Yaskawa INFORM job: SKRZYNIA_5240_0_STOPNI_2OBR.JBI

/JOB
//NAME SKRZYNIA_5240_0_STOPNI_2OBR
///FOLDERNAME 02-SKRZYNIE_JOBS
//POS
///NPOS 621,621,0,54,0,0
///TOOL 0
///POSTYPE PULSE
///PULSE
C00000=1055,-24125,84372,288,19725,204
C00001=0,-15438,65714,0,-68532,0
C00002=4718,-16587,59952,3396,-65485,-935
C00003=32997,-21499,42555,27623,-61436,21376
C00004=31759,-20688,42932,26837,-60850,21559
C00005=28987,-21156,42712,24818,-60442,22222
C00006=33447,-21964,42352,27886,-61721,21330
C00007=37687,-23357,41794,30651,-63289,20620
C00008=38979,-19018,48057,32961,-64962,20678
C00009=37261,-18075,48526,31902,-64209,20901
C00010=35830,-17198,48994,31015,-63571,21092
C00011=34080,-17614,48768,29780,-63290,21485
C00012=37261,-18075,48526,31902,-64209,20901
C00013=47373,-21912,40596,41149,-66086,26950
C00014=0,-15438,65714,0,-68532,0
C00015=4718,-16587,59952,3396,-65485,-935
C00016=32997,-21499,42555,27623,-61436,21376
C00017=31759,-20688,42932,26837,-60850,21559
C00018=28987,-21156,42712,24818,-60442,22222
C00019=33447,-21964,42352,27886,-61721,21330
C00020=37687,-23357,41794,30651,-63289,20620
C00021=38979,-19018,48057,32961,-64962,20678
C00022=37261,-18075,48526,31902,-64209,20901
C00023=35830,-17198,48994,31015,-63571,21092
C00024=34080,-17614,48768,29780,-63290,21485
C00025=37261,-18075,48526,31902,-64209,20901
C00026=47373,-21912,40596,41149,-66086,26950
C00027=45033,-20851,41104,39798,-65001,27223
C00028=42790,-19693,41704,38494,-63946,27495
C00029=41070,-20182,41442,37324,-63566,27891
C00030=45033,-20851,41104,39798,-65001,27223
C00031=45033,-20851,41104,39798,-65001,27223
C00032=59624,-29540,14278,64846,-60867,16042
C00033=57357,-28542,14780,63940,-59509,16120
C00034=56188,-29140,14476,63237,-58995,16387
C00035=59588,-29370,14363,64862,-60819,16012
C00036=62924,-29779,15793,65870,-63073,16252
C00037=59724,-28781,16276,64511,-61238,16415
C00038=57764,-27936,16704,63709,-60078,16488
C00039=56408,-28589,16373,62897,-59486,16787
C00040=59724,-28781,16276,64511,-61238,16415
C00041=87562,-48087,-13810,78020,-75252,11220
C00042=10104,-46603,4759,11228,-37390,-5046
C00043=0,-52280,40443,0,6876,0
C00044=1529,-42140,58025,-5964,2417,3265
C00045=0,-38374,23626,-1605,-51738,268
C00046=45044,-23015,37260,35797,-71879,25522
C00047=39973,-29571,18873,35060,-63052,24165
C00048=38620,-28701,19269,34339,-62304,24363
C00049=36409,-29254,19014,32896,-61805,24958
C00050=44451,-29039,21934,37281,-65892,23702
C00051=49472,-39353,6917,53118,-50908,20251
C00052=45058,-39356,3832,51653,-47640,20099
C00053=42883,-38319,4163,50577,-46309,20295
C00054=40255,-38926,3967,48502,-45334,21060
C00055=46774,-39679,3737,52663,-48537,19827
C00056=48708,-40455,3517,53615,-49689,19657
C00057=43798,-39237,3871,50850,-47027,20335
C00058=41951,-38324,4161,49930,-45891,20507
C00059=39836,-38844,3994,48234,-45126,21137
C00060=48489,-40338,3551,53521,-49551,19665
C00061=48489,-40338,3551,53521,-49551,19665
C00062=44432,-39026,3936,51363,-47247,20139
C00063=42487,-38069,4248,50403,-46050,20315
C00064=39061,-38795,4009,47695,-44769,21310
C00065=44432,-39026,3936,51363,-47247,20139
C00066=45358,-49480,-3557,50155,-49322,21260
C00067=1817,-44984,2816,-3462,-45659,1296
C00068=1445,-28771,30219,-502,-63201,-220
C00069=1148,-56354,34370,-22,3827,-10
C00070=0,-52280,40443,0,6876,0
C00071=0,-49898,44897,0,-65513,0
C00072=52002,-27630,35066,40617,-70496,28619
C00073=38179,-24916,32897,32855,-63545,30206
C00074=36484,-23889,33369,31863,-62698,30449
C00075=33804,-24434,33113,30025,-62179,31112
C00076=38179,-24916,32897,32855,-63545,30206
C00077=78369,-41260,16071,67181,-65880,21417
C00078=38179,-24916,32897,32855,-63545,30206
C00079=36484,-23889,33369,31863,-62698,30449
C00080=33804,-24434,33113,30025,-62179,31112
C00081=38179,-24916,32897,32855,-63545,30206
C00082=42162,-28027,28994,48933,-45818,24803
C00083=39537,-27148,29331,47235,-44522,25156
C00084=37690,-27578,29159,45634,-43962,25669
C00085=41496,-28393,28854,48300,-45677,25033
C00086=137,-45861,52341,97,-67596,-14
C00087=-31499,-58302,-23356,15027,12889,-13082
C00088=-52768,-43016,-26078,18373,38595,-18774
C00089=-89470,-32103,-32973,29905,69139,-31512
C00090=-68838,-26884,-24872,16972,64732,-23076
C00091=-53036,-11528,-12218,12363,64665,-17409
C00092=-51536,-9474,-10276,11905,64649,-16876
C00093=-51739,-9114,-7787,12104,63269,-17104
C00094=-53036,-11528,-12218,12363,64665,-17409
C00095=-17541,-26226,-24397,927,59032,-5038
C00096=-17541,-26226,-24397,927,59032,-5038
C00097=-16950,-23991,-22741,715,59568,-4818
C00098=-17036,-23563,-20101,755,58071,-4857
C00099=-17541,-26226,-24397,927,59032,-5038
C00100=34102,-23192,-21614,-15638,64271,13209
C00101=33423,-21885,-20599,-15423,64418,12942
C00102=32426,-19856,-18975,-15106,64629,12551
C00103=32578,-19611,-17013,-15290,63535,12762
C00104=33423,-21885,-20599,-15423,64418,12942
C00105=59339,-6070,-6417,-20979,72191,20891
C00106=59339,-6070,-6417,-20979,72191,20891
C00107=57897,-4256,-4562,-20702,71913,20431
C00108=58108,-3992,-2506,-20878,70835,20713
C00109=59339,-6070,-6417,-20979,72191,20891
C00110=42744,-35904,-30225,-18322,62562,16651
C00111=-53036,-11528,-12218,12363,64665,-17409
C00112=-77982,-26538,-29134,27151,66629,-27745
C00113=-70983,-8594,-1966,26503,59809,-49670
C00114=-80152,19776,40785,37351,72704,-50428
C00115=-79984,20154,42529,37516,71911,-50638
C00116=-79233,18397,40079,37458,71885,-50340
C00117=-79984,20154,42529,37516,71911,-50638
C00118=-73519,23289,38838,28890,77081,-45618
C00119=-73519,24511,42682,29072,75582,-46027
C00120=-73519,23289,38838,28890,77081,-45618
C00121=-88897,15706,42282,50101,71325,-56974
C00122=-88897,15706,42282,50101,71325,-56974
C00123=-87612,12343,37838,50071,70996,-56519
C00124=-85283,14202,40272,50301,69633,-56165
C00125=-87338,12550,38107,50098,70839,-56476
C00126=-84952,-1789,13569,34660,47724,-58955
C00127=-67641,-1674,11109,10330,44856,-44725
C00128=-66443,961,13975,9688,44721,-44210
C00129=-67641,-1674,11109,10330,44856,-44725
C00130=-67641,-376,15347,10694,42950,-44967
C00131=-67641,-1674,11109,10330,44856,-44725
C00132=-79040,417,20398,15965,28992,-57786
C00133=-76655,5212,30978,15501,25024,-57306
C00134=-76655,6949,35816,16758,23084,-57955
C00135=-76655,5212,30978,15501,25024,-57306
C00136=-74761,6919,33010,13466,24593,-56049
C00137=-80460,-2874,12270,15804,32253,-57809
C00138=-61258,-29124,-13156,26560,43617,-22150
C00139=-30420,-40507,-29240,27153,53235,15188
C00140=-18589,-38725,-21450,23338,47896,18931
C00141=-17722,-35233,-16455,23322,46926,19051
C00142=-17722,-33749,-12435,23948,45421,18620
C00143=-17722,-33892,-12819,23887,45564,18661
C00144=-16677,-31133,-11209,23138,46167,19311
C00145=-17819,-35820,-17540,23246,47228,19090
C00146=-74104,-11494,-6266,31916,75042,4269
C00147=-71226,-7329,2631,32115,71468,4273
C00148=-71226,-6504,5446,32343,70365,3922
C00149=-71226,-6611,5086,32313,70505,3967
C00150=-68386,-4058,7675,32040,69573,4789
C00151=-73314,-9412,-353,32206,72648,3829
C00152=51751,-31069,-22965,-10739,49070,48663
C00153=49028,-23852,-11575,-9841,46366,47823
C00154=49028,-23004,-8935,-10039,45204,47956
C00155=49028,-23118,-9286,-10013,45357,47939
C00156=47000,-20813,-7527,-8928,45644,47024
C00157=50476,-26208,-15307,-10408,47325,48332
C00158=90602,-5375,6902,-38786,69848,59444
C00159=83174,19950,50269,-44999,67580,58220
C00160=82362,17902,47383,-44926,67511,57879
C00161=83515,19072,48341,-44798,68200,58056
C00162=78091,19382,40247,-36371,72286,52960
C00163=78091,20664,44011,-36670,70997,53443
C00164=78091,19382,40247,-36371,72286,52960
C00165=88699,7296,38566,-55615,63182,60372
C00166=86803,3068,32674,-55410,62638,59657
C00167=84852,4315,34115,-55564,61561,59330
C00168=86803,3068,32674,-55410,62638,59657
C00169=92770,-2803,21719,-53893,67577,59421
C00170=73393,-10627,10934,-27897,30744,62458
C00171=70789,-6606,18800,-27824,27830,62140
C00172=69654,-4593,20814,-26755,27596,61444
C00173=70789,-6606,18800,-27824,27830,62140
C00174=70789,-5070,23059,-29482,26284,63017
C00175=70789,-6606,18800,-27824,27830,62140
C00176=83486,-8736,6503,-27040,35338,66550
C00177=77831,-2041,26192,-25270,18452,68895
C00178=77967,1961,32070,-26860,17569,69698
C00179=77967,5243,40752,-32914,14549,72656
C00180=77967,1961,32070,-26860,17569,69698
C00181=74560,4730,35257,-21622,16551,66717
C00182=77967,1961,32070,-26860,17569,69698
C00183=81109,-22356,2664,-22493,33121,60116
C00184=86168,-49730,-13668,-23926,46819,49343
C00185=44183,-52048,-7537,-24795,46064,51426
C00186=0,-52280,40443,0,6876,0
C00187=0,-52280,40443,0,6876,0
C00188=33629,-57276,-6399,46271,-24969,-2804
C00189=75493,-63502,-64712,103874,-64610,-6298
C00190=47968,-58405,-62693,109749,-46222,-10681
C00191=44214,-60060,-65896,114303,-43519,-9276
C00192=55379,-67378,-68041,108237,-48773,-4935
C00193=62671,-64213,-64640,104431,-56093,-7372
C00194=28458,-50318,6850,47420,-25887,-3347
C00195=0,-52280,40443,0,6876,0
C00196=1055,-24125,84372,288,19725,204
C00197=0,-15438,65714,0,-68532,0
C00198=0,-15438,65714,966,-70097,42926
C00199=69988,-9219,57065,61610,-82752,27767
C00200=63113,-6157,59685,58080,-79692,28271
C00201=46309,-5455,68070,40267,-75151,29719
C00202=49471,-5188,67710,43421,-76082,29577
C00203=63113,-6157,59685,58080,-79692,28271
C00204=69988,-9219,57065,61610,-82752,27767
C00205=0,-15438,65714,966,-70097,42926
C00206=0,-15438,65714,0,-68532,0
C00207=1055,-24125,84372,288,19725,204
C00208=1055,-24125,84372,288,19725,204
C00209=0,-52280,40443,0,6876,0
C00210=0,-17525,61946,0,273,32004
C00211=54446,-4421,37881,-48560,57645,57448
C00212=45059,-5790,38757,-53071,45868,54447
C00213=47134,-4843,57045,-85936,40972,71741
C00214=45953,-34,57521,-69944,42466,59819
C00215=35351,-3283,34371,-39408,48185,38080
C00216=43067,2853,36106,-38598,60324,43004
C00217=45059,-5790,38757,-53071,45868,54447
C00218=54446,-4421,37881,-48560,57645,57448
C00219=0,-17525,61946,0,273,32004
C00220=0,-52280,40443,0,6876,0
C00221=0,-52280,40443,0,6876,0
C00222=0,-52280,40443,0,6876,0
C00223=0,-52280,40443,0,-42737,40640
C00224=0,-52280,40443,0,-42737,40640
C00225=64551,-35409,28076,75550,-44539,17239
C00226=49799,-25338,45366,61341,-39751,21495
C00227=45731,-22710,35392,68644,-36821,18294
C00228=37964,-27036,25793,58834,-36141,20634
C00229=39068,-21674,37860,55103,-38849,23155
C00230=43117,-27612,29118,67655,-35359,18183
C00231=39863,-22026,47404,54615,-35502,22403
C00232=0,-52277,40442,0,6872,2
C00233=0,-38538,66749,0,-898,0
C00234=0,-52280,40443,0,-79033,35417
C00235=46775,-35113,22190,42926,-67531,20697
C00236=52587,-26056,25345,47610,-66542,17970
C00237=46075,-25504,24484,44216,-63256,18807
C00238=46254,-27712,19552,44922,-62123,18131
C00239=53914,-29436,22058,48262,-67266,17843
C00240=63113,-6157,59685,58080,-79692,28271
C00241=47789,-6280,67353,41142,-75661,29541
C00242=46856,-5642,67903,40595,-75324,29647
C00243=49490,-5202,67729,43369,-76086,29558
C00244=59203,-5425,63284,53118,-78384,28542
C00245=46775,-35113,22190,42926,-67531,20697
C00246=0,-52280,40443,0,-79033,35417
C00247=0,-52280,40443,0,-61239,28081
C00248=53819,-14110,13758,-46164,60155,50576
C00249=48398,-14119,9451,-44868,59619,48162
C00250=41138,-18250,21501,-61067,39474,53197
C00251=26203,-21075,4650,-31160,41208,31784
C00252=48398,-14119,9451,-44868,59619,48162
C00253=53819,-14110,13758,-46164,60155,50576
C00254=0,-52280,40443,0,-61239,28081
C00255=404,-42897,57020,-1574,2523,869
C00256=0,-52280,40443,0,6876,0
C00257=-99253,-13690,44082,59847,13407,-31313
C00258=-87814,-12734,20141,45739,-14352,-64418
C00259=-86669,-6582,30812,41148,-16781,-62025
C00260=-85055,-5827,31548,44003,-17420,-63187
C00261=-85971,-6262,31124,42409,-17052,-62539
C00262=-86650,-5303,32069,41395,-16716,-62141
C00263=-94954,-14494,-1860,-7818,15857,-59130
C00264=-94509,1544,30797,-849,15127,-60471
C00265=-94509,4151,37772,-1041,12286,-60378
C00266=-85971,-6262,31124,42409,-17052,-62539
C00267=-86125,-12470,22545,29004,-25567,-58412
C00268=-83883,-11340,22525,32952,-25567,-60136
C00269=-82768,-10824,22986,34487,-25904,-60776
C00270=-83883,-11340,22525,32952,-25567,-60136
C00271=-85143,-9772,23941,31487,-24966,-59556
C00272=-83883,-11340,22525,32952,-25567,-60136
C00273=-85732,-21202,11427,30682,-24763,-59235
C00274=-84150,-10929,23786,31981,-25941,-59678
C00275=-83036,-10419,24246,33504,-26268,-60308
C00276=-84150,-10929,23786,31981,-25941,-59678
C00277=-85291,-9507,25078,30650,-25411,-59154
C00278=-84150,-10929,23786,31981,-25941,-59678
C00279=-85786,-16909,14677,31743,-23900,-59790
C00280=-84150,-10498,24888,31517,-26306,-59436
C00281=-83174,-10052,25293,32841,-26587,-59984
C00282=-84150,-10498,24888,31517,-26306,-59436
C00283=-85258,-9112,26156,30226,-25800,-58928
C00284=-84150,-10498,24888,31517,-26306,-59436
C00285=-87841,-18519,13420,28367,-23534,-58339
C00286=-85040,-10859,24618,30253,-26091,-58908
C00287=-83241,-10052,25348,32714,-26598,-59924
C00288=-84150,-10465,24972,31484,-26336,-59417
C00289=-85145,-9228,26102,30329,-25881,-58963
C00290=-84150,-10465,24972,31484,-26336,-59417
C00291=-86371,-18277,13606,30568,-23951,-59265
C00292=-84345,-11688,21985,32461,-25312,-59957
C00293=-83211,-11173,22442,34044,-25650,-60618
C00294=-84345,-11688,21985,32461,-25312,-59957
C00295=-85283,-10526,23025,31366,-24861,-59525
C00296=-84345,-11688,21985,32461,-25312,-59957
C00297=-86191,-19647,12567,30467,-24278,-59187
C00298=-84345,-10877,24073,31552,-26006,-59481
C00299=-83051,-10286,24607,33321,-26381,-60213
C00300=-84345,-10877,24073,31552,-26006,-59481
C00301=-85179,-9842,25009,30582,-25619,-59100
C00302=-84345,-10877,24073,31552,-26006,-59481
C00303=-85438,-18022,14839,31140,-24818,-59429
C00304=-84247,-11820,22550,32049,-25753,-59727
C00305=-84104,-10976,23642,32111,-25899,-59738
C00306=-82990,-10465,24105,33639,-26227,-60372
C00307=-84104,-10976,23642,32111,-25899,-59738
C00308=-84898,-9998,24525,31196,-25529,-59378
C00309=-84104,-10976,23642,32111,-25899,-59738
C00310=-86610,-16845,14732,30573,-23614,-59301
C00311=-84104,-10864,23927,31990,-25993,-59674
C00312=-82824,-10273,24459,33737,-26370,-60397
C00313=-84104,-10864,23927,31990,-25993,-59674
C00314=-84789,-10021,24690,31200,-25673,-59363
C00315=-84104,-10864,23927,31990,-25993,-59674
C00316=-83806,-19585,12613,33764,-25080,-60559
C00317=-83924,-10205,25475,31619,-26533,-59453
C00318=-82780,-9675,25960,33156,-26866,-60087
C00319=-83924,-10205,25475,31619,-26533,-59453
C00320=-84478,-9530,26093,30986,-26280,-59206
C00321=-83924,-10205,25475,31619,-26533,-59453
C00322=-87149,-17993,13826,29513,-23647,-58830
C00323=-84920,-13182,20975,31162,-25481,-59361
C00324=-83711,-10572,24852,32056,-26475,-59649
C00325=-82779,-10142,25241,33309,-26748,-60166
C00326=-83711,-10572,24852,32056,-26475,-59649
C00327=-84370,-9774,25579,31305,-26170,-59356
C00328=-83711,-10572,24852,32056,-26475,-59649
C00329=-83642,-3679,42021,23358,-36761,-56118
C00330=-85886,-5975,41264,18964,-40261,-54782
C00331=-83919,-11632,22322,32811,-25616,-60079
C00332=-82884,-11162,22742,34234,-25925,-60671
C00333=-83919,-11632,22322,32811,-25616,-60079
C00334=-84723,-10654,23196,31887,-25230,-59715
C00335=-83919,-11632,22322,32811,-25616,-60079
C00336=-87348,-16035,7353,17528,-35245,-56477
C00337=-86244,-15062,8172,18754,-35315,-57058
C00338=-86244,-16649,3638,19674,-33501,-57585
C00339=-85308,-16228,3988,20718,-33648,-58082
C00340=-86244,-16649,3638,19674,-33501,-57585
C00341=-86740,-15973,4201,19194,-33277,-57362
C00342=-86244,-16649,3638,19674,-33501,-57585
C00343=-73780,-8639,20128,34258,-51705,-52097
C00344=-90711,-17528,-28778,11328,-28245,-57111
C00345=-92565,-19610,-33223,7138,-24591,-57051
C00346=-91512,-19116,-32812,8551,-24603,-57834
C00347=-92565,-19610,-33223,7138,-24591,-57051
C00348=-93003,-18716,-32476,6600,-24397,-56752
C00349=-92565,-19610,-33223,7138,-24591,-57051
C00350=-92565,-19610,-33223,7138,-24591,-57051
C00351=-95836,-54375,-51122,6031,-17685,-48210
C00352=-95836,-54375,-51122,6031,-17685,-48210
C00353=-43821,-47238,-2775,-3022,56549,-3681
C00354=-20126,-26882,59542,2406,16879,-9162
C00355=-20126,-26882,59542,2406,16879,-9162
C00356=98601,-10520,92678,4674,-40855,-9615
C00357=95537,-19831,-2695,-2933,-44471,35837
C00358=92548,-20391,-28429,-6186,-30623,55200
C00359=91429,-17018,-28974,-8057,-27827,56250
C00360=91429,-17018,-28974,-8057,-27827,56250
C00361=90371,-16495,-28521,-9286,-27856,56953
C00362=91429,-17018,-28974,-8057,-27827,56250
C00363=92033,-15799,-27911,-7415,-27588,55880
C00364=91429,-17018,-28974,-8057,-27827,56250
C00365=92548,-20391,-28429,-6186,-30623,55200
C00366=91156,-15018,-4648,-8036,-38181,54813
C00367=90585,-14766,-4428,-8565,-38201,55100
C00368=88830,-13959,-3717,-10186,-38284,55977
C00369=89897,-14456,-4157,-9202,-38230,55445
C00370=90761,-12944,-2809,-8452,-37927,55043
C00371=89897,-14456,-4157,-9202,-38230,55445
C00372=89910,-11217,67535,-9455,-58896,55399
C00373=89910,-11217,67535,-9455,-58896,55399
C00374=85786,-16735,14816,-31782,-23869,59812
C00375=83514,-12996,17929,-35760,-24132,61552
C00376=82251,-12406,18443,-37550,-24551,62308
C00377=83514,-12996,17929,-35760,-24132,61552
C00378=84258,-12095,18717,-34917,-23742,61217
C00379=83514,-12996,17929,-35760,-24132,61552
C00380=87149,-17993,13826,-29513,-23647,58830
C00381=83118,-12818,18089,-36330,-24263,61791
C00382=81915,-12248,18589,-38020,-24666,62504
C00383=83118,-12818,18089,-36330,-24263,61791
C00384=83897,-11882,18912,-35460,-23856,61445
C00385=83118,-12818,18089,-36330,-24263,61791
C00386=83806,-19585,12613,-33764,-25080,60559
C00387=82998,-13006,17925,-36445,-24332,61826
C00388=81675,-12378,18472,-38297,-24777,62607
C00389=82998,-13006,17925,-36445,-24332,61826
C00390=83876,-11958,18841,-35466,-23874,61442
C00391=82998,-13006,17925,-36445,-24332,61826
C00392=86610,-16845,14732,-30573,-23614,59301
C00393=82493,-13239,17725,-37070,-24559,62089
C00394=81406,-12724,18174,-38578,-24928,62723
C00395=82493,-13239,17725,-37070,-24559,62089
C00396=83436,-12134,18690,-36041,-24064,61684
C00397=82493,-13239,17725,-37070,-24559,62089
C00398=84814,-16043,15376,-33312,-24093,60464
C00399=82555,-13613,17404,-36910,-24580,62015
C00400=81384,-13062,17878,-38534,-24974,62698
C00401=82555,-13613,17404,-36910,-24580,62015
C00402=83566,-12434,18427,-35805,-24047,61580
C00403=82555,-13613,17404,-36910,-24580,62015
C00404=86191,-19647,12567,-30467,-24278,59187
C00405=82500,-13648,17375,-36975,-24607,62039
C00406=81467,-13161,17792,-38413,-24955,62645
C00407=82500,-13648,17375,-36975,-24607,62039
C00408=83481,-12505,18364,-35905,-24087,61617
C00409=82500,-13648,17375,-36975,-24607,62039
C00410=86371,-18277,13606,-30568,-23951,59265
C00411=82904,-13790,17251,-36416,-24470,61808
C00412=81715,-13237,17726,-38081,-24865,62509
C00413=82904,-13790,17251,-36416,-24470,61808
C00414=83686,-12878,18037,-35556,-24055,61469
C00415=82904,-13790,17251,-36416,-24470,61808
C00416=87841,-18519,13420,-28367,-23534,58339
C00417=83645,-14279,16834,-35321,-24258,61342
C00418=81692,-13388,17594,-38077,-24893,62505
C00419=82748,-13879,17174,-36603,-24542,61883
C00420=83607,-12881,18032,-35663,-24082,61515
C00421=82748,-13879,17174,-36603,-24542,61883
C00422=85786,-16909,14677,-31743,-23900,59790
C00423=83053,-14438,16700,-36077,-24500,61654
C00424=81460,-13708,17319,-38301,-25026,62591
C00425=82520,-14198,16902,-36833,-24674,61972
C00426=83571,-12989,17938,-35691,-24113,61524
C00427=82520,-14198,16902,-36833,-24674,61972
C00428=85732,-21202,11427,-30682,-24763,59235
C00429=82985,-14628,16542,-36121,-24556,61664
C00430=81172,-13798,17245,-38643,-25153,62725
C00431=82398,-14365,16763,-36952,-24745,62014
C00432=83600,-12984,17944,-35650,-24102,61504
C00433=82398,-14365,16763,-36952,-24745,62014
C00434=92346,-18713,13565,-21110,-22545,55257
C00435=83441,-14269,16838,-35588,-24331,61454
C00436=81518,-13384,17592,-38292,-24965,62594
C00437=82794,-13980,17083,-36511,-24538,61844
C00438=83714,-12912,18003,-35501,-24048,61445
C00439=82794,-13980,17083,-36511,-24538,61844
C00440=86642,-13028,12466,-93429,-10417,85802
C00441=86140,-12802,12665,-93523,-10743,85795
C00442=85030,-12289,13120,-93723,-11463,85776
C00443=86140,-12802,12665,-93523,-10743,85795
C00444=86958,-11660,13681,-94506,-10238,86349
C00445=85239,-16743,-4327,42764,21357,45785
C00446=86674,107,23869,25042,24033,51593
C00447=86674,2327,30134,27824,21680,50173
C00448=86140,-12802,12665,-93523,-10743,85795
C00449=85045,-36869,-4353,-28502,-22832,52282
C00450=0,-24029,84339,0,19981,0
C00451=0,-24029,84339,0,19981,0
C00452=3172,-24246,80980,3465,15913,689
C00453=-86563,-26985,13879,10257,-21548,-45530
C00454=-86191,-19647,12567,30467,-24278,-59187
C00455=-83221,-13587,17636,37793,-25116,-62228
C00456=-91978,-13833,14560,12391,-18633,-51524
C00457=-94992,-13830,14285,1276,-18012,-46664
C00458=-84074,-17488,11256,38660,-23649,-62784
C00459=-73679,-33270,1000,44272,-31600,-64253
C00460=-86926,-60758,23267,6576,1160,-9545
C00461=0,-52280,40443,0,6876,0
C00462=82475,-58079,26734,835,4084,4444
C00463=97932,-26840,7691,8784,-23444,42538
C00464=87166,-16607,16322,-25365,-24201,56345
C00465=84699,-11354,21752,-29145,-24735,57949
C00466=84804,-11023,22730,-28561,-25071,57659
C00467=85100,-26994,10417,-24982,-28140,55821
C00468=0,-52280,40443,0,6876,0
C00469=0,-52280,40443,0,6876,0
C00470=-90140,-60305,18108,-2708,1721,-7625
C00471=-95594,-27428,6866,-4663,-19832,-42154
C00472=-98688,-13767,16447,-18366,-10080,-35766
C00473=-98964,-4977,31041,-27811,-8682,-30400
C00474=-98987,-3006,34487,-29035,-8628,-29652
C00475=-100063,5316,51567,-32262,-10006,-27560
C00476=-94446,19117,65275,-6998,10272,-43293
C00477=-95535,2380,25473,239,27557,-47214
C00478=-91562,2960,34279,-4747,22029,-44179
C00479=-95534,12584,45578,298,21393,-47243
C00480=-99268,-13088,27343,-18620,-14105,-35021
C00481=-90140,-60305,18108,-2708,1721,-7625
C00482=0,-52280,40443,0,6876,0
C00483=84259,-57935,27522,-3761,3673,6310
C00484=86507,-39672,4297,-27618,-16640,46340
C00485=73669,-37119,-20783,-92053,-19719,85232
C00486=86539,-20830,1725,-71850,-11773,76853
C00487=94927,-16191,10904,-46169,-1414,61414
C00488=97704,-11547,13178,-56709,4181,66931
C00489=98315,-9028,11559,-15530,14603,48461
C00490=96173,-949,20667,-3174,24056,38215
C00491=95132,-6008,10010,1655,28777,36730
C00492=94050,-4358,6626,-2469,41779,36653
C00493=97858,4348,15692,-4839,42267,38390
C00494=100487,-9453,-1206,-10413,41328,41147
C00495=96250,-19428,-8283,-4838,27297,37910
C00496=86507,-39672,4297,-27618,-16640,46340
C00497=84259,-57935,27522,-3761,3673,6310
C00498=0,-52280,40443,0,6876,0
C00499=0,-27933,77061,0,20812,0
C00500=0,-27933,77061,0,20812,0
C00501=0,-52280,40443,0,6876,0
C00502=-91970,-60791,14435,-3343,512,-9412
C00503=-98647,-24138,10005,-11519,-21203,-39749
C00504=-99883,-13980,22886,-11640,-25090,-40341
C00505=-99702,-9154,61728,-1148,-61809,-40243
C00506=-84328,-13042,29707,23458,-33731,-54641
C00507=-83101,-4179,39208,25894,-34785,-55667
C00508=-82881,-4330,38692,26392,-34479,-55866
C00509=-76259,-18287,26646,31659,-38322,-57579
C00510=-89741,-28009,12101,4461,-28076,-46404
C00511=-91970,-60791,14435,-3343,512,-9412
C00512=0,-52280,40443,0,6876,0
C00513=91083,-60784,14823,-9043,-825,15173
C00514=83869,-19403,12921,-33769,-24740,60260
C00515=83869,-19403,12921,-33769,-24740,60260
C00516=83932,-19538,53415,-33663,-71112,60249
C00517=83932,-19538,53415,-33663,-71112,60249
C00518=82480,-12247,21118,-35440,-26416,60009
C00519=82194,-11433,19802,-37650,-25323,61125
C00520=81904,-9374,24711,-35791,-26879,60109
C00521=79790,-20261,14917,-36681,-28829,60258
C00522=76554,-29711,-1870,-46042,-25952,65654
C00523=91083,-60784,14823,-9043,-825,15173
C00524=0,-52280,40443,0,6876,0
C00525=-91526,-60598,16699,7584,176,-13289
C00526=-81382,-25890,9219,35455,-25500,-59095
C00527=-86453,-20958,12525,30076,-22568,-57089
C00528=-86589,-16097,16237,31250,-21582,-57704
C00529=-98933,-11298,20505,-13970,-18736,-37953
C00530=-98281,-10965,21163,-11559,-18548,-39330
C00531=-85424,-18472,14402,34409,-22969,-58895
C00532=-74746,-27148,8488,44263,-29128,-62418
C00533=-81326,-27507,8265,35533,-26282,-59001
C00534=-91415,-60262,16631,7870,-73,-13734
C00535=24,-24029,84339,7,19981,5
C00536=100404,-52373,45687,-1822,14816,-5144
C00537=75939,-26469,7919,-40869,-29645,63133
C00538=81882,-22565,10470,-35355,-26404,61107
C00539=82801,-12246,21732,-34208,-26055,60642
C00540=91844,-10818,23389,-8611,-22226,49798
C00541=96558,-9677,26191,5829,-23135,43648
C00542=77262,-23244,14300,-38922,-31295,61912
C00543=78410,-22868,15324,-38001,-30064,61274
C00544=96357,-33562,33410,58602,-23427,10353
C00545=568,-24029,84339,168,19981,112
C00546=-91970,-60791,14435,-3343,512,-9412
C00547=-98991,-22833,11519,-12824,-17638,-36336
C00548=-86376,-13627,18436,38326,-18406,-58533
C00549=-85581,-10814,20279,41280,-18093,-59893
C00550=-85551,-10406,21021,40925,-18257,-59713
C00551=-86274,-24518,9978,34497,-20333,-56613
C00552=-91684,-53777,2301,20525,-9313,-33684
C00553=-67305,-55044,34987,1504,5690,-2468
C00554=0,-52280,40443,0,6876,0
C00555=77036,-56616,31288,-2531,4707,4197
C00556=84359,-28321,8817,-32860,-20485,54199
C00557=81156,-16932,14874,-39538,-26422,62851
C00558=93122,-15135,13007,-5735,-18111,48773
C00559=90767,-14192,15510,-13532,-19632,52035
C00560=77970,-27630,4721,-41834,-28549,63607
C00561=81111,-35571,7141,-33980,-21909,52006
C00562=82626,-57814,28323,-4146,3364,6346
C00563=0,-52280,40443,0,6876,0
C00564=0,-28135,76691,0,20839,0
C00565=0,-28135,76691,0,20839,0
C00566=-45332,-39712,59352,-1730,18713,2903
C00567=-94065,-8316,59352,-1730,-37754,-40387
C00568=-100331,-14895,33931,-8215,-36518,-40227
C00569=-98931,-8578,39429,-6260,-48307,-43744
C00570=-100336,-4176,46216,-7600,-55875,-44633
C00571=-93952,8947,73671,995,-68520,-43850
C00572=-98791,-3170,32594,-4861,-60761,-43748
C00573=-98768,4156,37660,-4945,-58738,-43661
C00574=-98673,-12696,-17797,-7569,-33360,-41896
C00575=-99330,-14840,-29426,-9917,-27109,-40593
C00576=-99605,-15546,-21493,-8548,-33053,-41326
C00577=-100467,-8208,-2562,-8095,-44661,-42156
C00578=-93952,8947,73671,995,-68520,-43850
C00579=-88754,54,62805,4404,-67858,-45120
C00580=-100222,-4532,45667,-7492,-55263,-44561
C00581=-100331,-14895,33931,-8215,-36518,-40227
C00582=-94065,-8316,59352,-1730,-37754,-40387
C00583=-45544,-32973,71870,-2133,15168,3033
C00584=0,-28135,76691,0,20839,0
C00585=54178,-17846,77779,596,-29686,20997
C00586=54178,-17846,77779,596,-29686,20997
C00587=99462,-18987,75418,611,-28919,20989
C00588=98707,-9390,78674,1080,-71212,38250
C00589=98768,-5182,41096,1808,-44974,38308
C00590=100431,1771,51615,3823,-56746,39115
C00591=97953,-6621,17555,2289,-50176,39420
C00592=95834,-5353,18817,760,-50052,40242
C00593=86453,-3910,18511,-13431,-48443,44868
C00594=88887,-11110,-8515,-11527,-36861,46615
C00595=88808,-13839,-20865,-13699,-30585,47852
C00596=90457,-16080,-12990,-9972,-37305,45724
C00597=97953,-6621,17555,2289,-50176,39420
C00598=100431,1771,51615,3823,-56746,39115
C00599=98768,-5182,41096,1808,-44974,38308
C00600=98707,-9390,78674,1080,-71212,38250
C00601=0,-28135,76691,0,20839,0
C00602=0,-28135,76691,0,20839,0
C00603=-91526,-60598,16699,7584,176,-13289
C00604=-81382,-25890,9219,35455,-25500,-59095
C00605=-81382,-25890,9219,35455,-25500,-59095
C00606=-85509,-13950,19358,32213,-22393,-58041
C00607=-96341,-12086,19487,-5053,-17846,-42145
C00608=-97523,-9822,24708,-8570,-19966,-40659
C00609=-84656,-25369,12054,31249,-26195,-57129
C00610=-82652,-57346,29982,2770,3944,-5064
C00611=0,-52280,40443,0,6876,0
C00612=60653,-54633,35892,-1212,5841,2035
C00613=77942,-28227,6869,-38010,-29303,61907
C00614=82500,-13648,17375,-36975,-24607,62039
C00615=80731,-11587,18684,-41654,-25449,63953
C00616=80409,-10373,22284,-40214,-26848,63104
C00617=64389,-31987,5108,-50419,-37074,66126
C00618=60653,-54633,35892,-1212,5841,2035
C00619=0,-52280,40443,0,6876,0
C00620=0,-28167,76633,0,20843,0
BC00000=413138
BC00001=413138
BC00002=295997
BC00003=264574
BC00004=264574
BC00005=264574
BC00006=264574
BC00007=233852
BC00008=284288
BC00009=284288
BC00010=284288
BC00011=284288
BC00012=284288
BC00013=356545
BC00014=413138
BC00015=388163
BC00016=356740
BC00017=356740
BC00018=356740
BC00019=356740
BC00020=356740
BC00021=407176
BC00022=407176
BC00023=407176
BC00024=407176
BC00025=407176
BC00026=479433
BC00027=479433
BC00028=479433
BC00029=479433
BC00030=479433
BC00031=530237
BC00032=530237
BC00033=530237
BC00034=530237
BC00035=530237
BC00036=601977
BC00037=601977
BC00038=601977
BC00039=601977
BC00040=601977
BC00041=601977
BC00042=522422
BC00043=522422
BC00044=671734
BC00045=689202
BC00046=689202
BC00047=689202
BC00048=689202
BC00049=689202
BC00050=689202
BC00051=726463
BC00052=726463
BC00053=726463
BC00054=726463
BC00055=726463
BC00056=782137
BC00057=782137
BC00058=782137
BC00059=782137
BC00060=782137
BC00061=850421
BC00062=850421
BC00063=850421
BC00064=850421
BC00065=850421
BC00066=850421
BC00067=823841
BC00068=797607
BC00069=755227
BC00070=755227
BC00071=915219
BC00072=914226
BC00073=914226
BC00074=914226
BC00075=914226
BC00076=914226
BC00077=914226
BC00078=983350
BC00079=983350
BC00080=983350
BC00081=983350
BC00082=963371
BC00083=963371
BC00084=963371
BC00085=963371
BC00086=922367
BC00087=927819
BC00088=927819
BC00089=927819
BC00090=943180
BC00091=943180
BC00092=943180
BC00093=943180
BC00094=943180
BC00095=943180
BC00096=943180
BC00097=943180
BC00098=943180
BC00099=943180
BC00100=943180
BC00101=943180
BC00102=943180
BC00103=943180
BC00104=943180
BC00105=943180
BC00106=943180
BC00107=943180
BC00108=943180
BC00109=943180
BC00110=943180
BC00111=943180
BC00112=943180
BC00113=943180
BC00114=943180
BC00115=943182
BC00116=943182
BC00117=943182
BC00118=943182
BC00119=943182
BC00120=943182
BC00121=943182
BC00122=943182
BC00123=943182
BC00124=943182
BC00125=943182
BC00126=943182
BC00127=943182
BC00128=943182
BC00129=943182
BC00130=943182
BC00131=943182
BC00132=943182
BC00133=943182
BC00134=943182
BC00135=943182
BC00136=943182
BC00137=943182
BC00138=943183
BC00139=943184
BC00140=943184
BC00141=943184
BC00142=943184
BC00143=943184
BC00144=943184
BC00145=943184
BC00146=943184
BC00147=943184
BC00148=943184
BC00149=943184
BC00150=943156
BC00151=943170
BC00152=943170
BC00153=943170
BC00154=943170
BC00155=943170
BC00156=943170
BC00157=943170
BC00158=943184
BC00159=943184
BC00160=943184
BC00161=943184
BC00162=943184
BC00163=943184
BC00164=943184
BC00165=943184
BC00166=943184
BC00167=943184
BC00168=943184
BC00169=943184
BC00170=943184
BC00171=943184
BC00172=943184
BC00173=943184
BC00174=943184
BC00175=943184
BC00176=943184
BC00177=943184
BC00178=943184
BC00179=943184
BC00180=943184
BC00181=943184
BC00182=943184
BC00183=911399
BC00184=884954
BC00185=838173
BC00186=838173
BC00187=727925
BC00188=734552
BC00189=750834
BC00190=750837
BC00191=811927
BC00192=811927
BC00193=760768
BC00194=744267
BC00195=744267
BC00196=413138
BC00197=413138
BC00198=413138
BC00199=408626
BC00200=408626
BC00201=408753
BC00202=347392
BC00203=408626
BC00204=408626
BC00205=413138
BC00206=413138
BC00207=413138
BC00208=505502
BC00209=697681
BC00210=697681
BC00211=733666
BC00212=758324
BC00213=766520
BC00214=794509
BC00215=817343
BC00216=794510
BC00217=758324
BC00218=733666
BC00219=697681
BC00220=697681
BC00221=697681
BC00222=841681
BC00223=841681
BC00224=884227
BC00225=901088
BC00226=895224
BC00227=896289
BC00228=924873
BC00229=947693
BC00230=921975
BC00231=887634
BC00232=824879
BC00233=507816
BC00234=507816
BC00235=552804
BC00236=552804
BC00237=551170
BC00238=493239
BC00239=491979
BC00240=285738
BC00241=285865
BC00242=285441
BC00243=256782
BC00244=258630
BC00245=552804
BC00246=507816
BC00247=507816
BC00248=507816
BC00249=531288
BC00250=531293
BC00251=591541
BC00252=531288
BC00253=507816
BC00254=507816
BC00255=507816
BC00256=848972
BC00257=861901
BC00258=963633
BC00259=963633
BC00260=963633
BC00261=963633
BC00262=963633
BC00263=963633
BC00264=963633
BC00265=963633
BC00266=963633
BC00267=963633
BC00268=963633
BC00269=963633
BC00270=963633
BC00271=963633
BC00272=963633
BC00273=902188
BC00274=895372
BC00275=895372
BC00276=895372
BC00277=895372
BC00278=895372
BC00279=840744
BC00280=840744
BC00281=840744
BC00282=840744
BC00283=840744
BC00284=840744
BC00285=779300
BC00286=771332
BC00287=771332
BC00288=771332
BC00289=771332
BC00290=771332
BC00291=717855
BC00292=717855
BC00293=717855
BC00294=717855
BC00295=717855
BC00296=717855
BC00297=656405
BC00298=649173
BC00299=649173
BC00300=649173
BC00301=649173
BC00302=649173
BC00303=594961
BC00304=594961
BC00305=594961
BC00306=594961
BC00307=594961
BC00308=594961
BC00309=594961
BC00310=533517
BC00311=525229
BC00312=525229
BC00313=525229
BC00314=525229
BC00315=525229
BC00316=472073
BC00317=472073
BC00318=472073
BC00319=472073
BC00320=472073
BC00321=472073
BC00322=410629
BC00323=405662
BC00324=402968
BC00325=402968
BC00326=402968
BC00327=402968
BC00328=402968
BC00329=402968
BC00330=349186
BC00331=349186
BC00332=349186
BC00333=349186
BC00334=349186
BC00335=349186
BC00336=336469
BC00337=336469
BC00338=336469
BC00339=336469
BC00340=336469
BC00341=336469
BC00342=336469
BC00343=367602
BC00344=367601
BC00345=367601
BC00346=367601
BC00347=367601
BC00348=367601
BC00349=367601
BC00350=425303
BC00351=425303
BC00352=514953
BC00353=463119
BC00354=419862
BC00355=484962
BC00356=484962
BC00357=395463
BC00358=369502
BC00359=369502
BC00360=369502
BC00361=369502
BC00362=369502
BC00363=369502
BC00364=369502
BC00365=369502
BC00366=368885
BC00367=368885
BC00368=368885
BC00369=368885
BC00370=368885
BC00371=368885
BC00372=419064
BC00373=366918
BC00374=349186
BC00375=353241
BC00376=353241
BC00377=353241
BC00378=353241
BC00379=353241
BC00380=410629
BC00381=409135
BC00382=409135
BC00383=409135
BC00384=409135
BC00385=409135
BC00386=472073
BC00387=476126
BC00388=476126
BC00389=476126
BC00390=476126
BC00391=476126
BC00392=533517
BC00393=532644
BC00394=532644
BC00395=532644
BC00396=532644
BC00397=532644
BC00398=594961
BC00399=599988
BC00400=599988
BC00401=599988
BC00402=599988
BC00403=599988
BC00404=656405
BC00405=653254
BC00406=653254
BC00407=653254
BC00408=653254
BC00409=653254
BC00410=717855
BC00411=721570
BC00412=721570
BC00413=721570
BC00414=721570
BC00415=721570
BC00416=779300
BC00417=777963
BC00418=777963
BC00419=777963
BC00420=777963
BC00421=777963
BC00422=840744
BC00423=843810
BC00424=843810
BC00425=843810
BC00426=843810
BC00427=843810
BC00428=902188
BC00429=900128
BC00430=900128
BC00431=900128
BC00432=900128
BC00433=900128
BC00434=963634
BC00435=965489
BC00436=965489
BC00437=965489
BC00438=965489
BC00439=965489
BC00440=965489
BC00441=965489
BC00442=965489
BC00443=965489
BC00444=965489
BC00445=965489
BC00446=965489
BC00447=965489
BC00448=965489
BC00449=931504
BC00450=769966
BC00451=769966
BC00452=716686
BC00453=679663
BC00454=721442
BC00455=721442
BC00456=721439
BC00457=781482
BC00458=781888
BC00459=781888
BC00460=781888
BC00461=781888
BC00462=768943
BC00463=718475
BC00464=718475
BC00465=718475
BC00466=778313
BC00467=778313
BC00468=717855
BC00469=792672
BC00470=792672
BC00471=948195
BC00472=948195
BC00473=957587
BC00474=959389
BC00475=967363
BC00476=950198
BC00477=956675
BC00478=956675
BC00479=956675
BC00480=950199
BC00481=792672
BC00482=792672
BC00483=792672
BC00484=887446
BC00485=956264
BC00486=956264
BC00487=969252
BC00488=969531
BC00489=979980
BC00490=973562
BC00491=973050
BC00492=971798
BC00493=971960
BC00494=956264
BC00495=956264
BC00496=887446
BC00497=792672
BC00498=792672
BC00499=700249
BC00500=546214
BC00501=546214
BC00502=546211
BC00503=546211
BC00504=406776
BC00505=406776
BC00506=352261
BC00507=346119
BC00508=406266
BC00509=406266
BC00510=491556
BC00511=546211
BC00512=546214
BC00513=546214
BC00514=507604
BC00515=410782
BC00516=429690
BC00517=375447
BC00518=350474
BC00519=350474
BC00520=408658
BC00521=408658
BC00522=507604
BC00523=546214
BC00524=546214
BC00525=516757
BC00526=591809
BC00527=591809
BC00528=591809
BC00529=591183
BC00530=650353
BC00531=650538
BC00532=650538
BC00533=584003
BC00534=515801
BC00535=520018
BC00536=520018
BC00537=590597
BC00538=593080
BC00539=593080
BC00540=593080
BC00541=652365
BC00542=652559
BC00543=594501
BC00544=537666
BC00545=433888
BC00546=546211
BC00547=830322
BC00548=830322
BC00549=830322
BC00550=890247
BC00551=890396
BC00552=798848
BC00553=798848
BC00554=798848
BC00555=798848
BC00556=832296
BC00557=845010
BC00558=845010
BC00559=904605
BC00560=904704
BC00561=818840
BC00562=818839
BC00563=818839
BC00564=526967
BC00565=334612
BC00566=334612
BC00567=334612
BC00568=350464
BC00569=350464
BC00570=359337
BC00571=359337
BC00572=359337
BC00573=359337
BC00574=359453
BC00575=359337
BC00576=359337
BC00577=359337
BC00578=359337
BC00579=359337
BC00580=358620
BC00581=350464
BC00582=334612
BC00583=334612
BC00584=334612
BC00585=334613
BC00586=501279
BC00587=501279
BC00588=334612
BC00589=334610
BC00590=349510
BC00591=365935
BC00592=365935
BC00593=365934
BC00594=348430
BC00595=348430
BC00596=348430
BC00597=365935
BC00598=349510
BC00599=334610
BC00600=334612
BC00601=334612
BC00602=512789
BC00603=516757
BC00604=526627
BC00605=466969
BC00606=466969
BC00607=466969
BC00608=524647
BC00609=525745
BC00610=525745
BC00611=525745
BC00612=525745
BC00613=473911
BC00614=473911
BC00615=473911
BC00616=532824
BC00617=533743
BC00618=525745
BC00619=525745
BC00620=525747
///POSTYPE BASE
///RECTAN
///RCONF 0,0,0,0,0,0,0,0,0,0,0,0,0,0,0,0,0,0,0,0,0,0,0,0
P00006=-2.449,0.031,8.825,0.0000,0.0000,0.0000
P00057=0.000,0.000,2.000,0.0000,0.0000,0.0000
P00058=0.000,0.000,3.000,0.0000,0.0000,0.0000
///RCONF 1,0,0,0,0,0,0,0,0,0,0,0,0,0,0,0,0,0,0,0,0,0,0,0
P00097=0.043,-1.896,1.568,0.0000,0.0000,0.0000
P00098=-0.089,-2.467,4.059,0.0000,0.0000,0.0000
P00099=0.011,-2.380,1.226,0.0000,0.0000,0.0000
P00100=-0.081,2.558,4.482,0.0000,0.0000,0.0000
P00101=0.030,-2.286,2.993,0.0000,0.0000,0.0000
P00102=-0.005,-1.108,1.644,0.0000,0.0000,0.0000
P00103=-0.094,-3.400,4.200,0.0000,0.0000,0.0000
P00104=0.043,-2.127,5.826,0.0000,0.0000,0.0000
P00105=-0.043,0.662,5.286,0.0000,0.0000,0.0000
P00106=-0.018,-2.519,0.237,0.0000,0.0000,0.0000
P00107=-0.008,-4.537,-4.500,0.0000,0.0000,0.0000
P00108=0.014,-3.040,2.637,0.0000,0.0000,0.0000
P00109=0.017,-3.622,2.341,0.0000,0.0000,0.0000
P00110=7346.140,158.997,-946.107,-0.1876,37.7131,-155.1643
///RCONF 0,0,0,0,0,0,0,0,0,0,0,0,0,0,0,0,0,0,0,0,0,0,0,0
P00299=-3.815,-1.565,6.918,0.0000,0.0000,0.0000
///RCONF 1,0,0,0,0,0,0,0,0,0,0,0,0,0,0,0,0,0,0,0,0,0,0,0
P00300=-0.036,-1.505,2.318,0.0000,0.0000,0.0000
///RCONF 0,0,0,0,0,0,0,0,0,0,0,0,0,0,0,0,0,0,0,0,0,0,0,0
P00301=0.005,-4.708,-4.628,0.0000,0.0000,0.0000
P00302=0.052,-2.937,-4.426,0.0000,0.0000,0.0000
P00303=-0.004,-1.437,-4.584,0.0000,0.0000,0.0000
P00304=0.028,-1.666,-4.234,0.0000,0.0000,0.0000
P00305=-0.003,-1.920,-3.501,0.0000,0.0000,0.0000
P00306=0.015,-2.252,-3.054,0.0000,0.0000,0.0000
P00307=0.019,-2.151,-5.077,0.0000,0.0000,0.0000
P00308=-0.003,-2.092,-4.888,0.0000,0.0000,0.0000
P00309=-0.040,-2.205,-4.992,0.0000,0.0000,0.0000
P00310=-0.006,-2.490,-5.925,0.0000,0.0000,0.0000
P00311=-0.007,-2.079,-5.307,0.0000,0.0000,0.0000
P00312=-0.032,2.202,-7.632,0.0000,0.0000,0.0000
///RCONF 1,0,0,0,0,0,0,0,0,0,0,0,0,0,0,0,0,0,0,0,0,0,0,0
P00349=0.060,0.167,-1.133,0.0000,0.0000,0.0000
///RCONF 0,0,0,0,0,0,0,0,0,0,0,0,0,0,0,0,0,0,0,0,0,0,0,0
P00350=11.519,-0.008,1.149,0.0000,0.0000,0.0000
P00351=13.563,-0.027,-0.653,0.0000,0.0000,0.0000
P00352=13.252,-0.027,-0.827,0.0000,0.0000,0.0000
P00353=10.971,-0.082,0.776,0.0000,0.0000,0.0000
P00354=-0.024,2.508,-1.824,0.0000,0.0000,0.0000
P00355=-0.001,2.528,-1.131,0.0000,0.0000,0.0000
P00356=-0.034,2.921,-0.262,0.0000,0.0000,0.0000
P00357=0.003,3.386,-0.091,0.0000,0.0000,0.0000
P00358=0.014,3.037,-0.020,0.0000,0.0000,0.0000
P00359=-0.005,2.731,0.912,0.0000,0.0000,0.0000
P00360=-0.011,3.412,0.438,0.0000,0.0000,0.0000
P00361=0.018,3.050,1.253,0.0000,0.0000,0.0000
P00362=0.014,2.784,0.148,0.0000,0.0000,0.0000
P00399=-2.449,0.031,8.825,0.0000,0.0000,0.0000
P00400=5.920,-3.503,-0.024,0.0000,0.0000,0.0000
P00401=3.430,-0.021,1.131,0.0000,0.0000,0.0000
P00402=-0.253,1.107,3.062,0.0000,0.0000,0.0000
P00403=-3.666,-0.015,5.328,0.0000,0.0000,0.0000
P00405=2.420,0.007,1.427,0.0000,0.0000,0.0000
P00406=3.513,-0.022,0.429,0.0000,0.0000,0.0000
P00415=-1.781,-1.303,3.250,0.0000,0.0000,0.0000
P00416=0.027,1.119,3.078,0.0000,0.0000,0.0000
//INST
///DATE 2025/03/06 15:39
///ATTR SC,RW
///GROUP1 RB1,BS1
NOP
CALL JOB:MOVE_INTO_TUNNEL
SFTOF
'------------------------
'------------------------
'SPOINA SRODEK DOL
'------------------------
'------------------------
MOVJ C00000 BC00000 VJ=10.00
MOVJ C00001 BC00001 VJ=30.00
'------------------------
'PODLOGA_BEZ_ROZPORKI
'------------------------
'TEST
MOVL C00002 BC00002 V=166.7
MOVL C00003 BC00003 V=166.7 PL=0
REFP 3 C00004 BC00004
CALL JOB:SEARCH-R1
IMOV P0057 V=23.0
SET P0097 P0006
SFTON P0097
REFP 3 C00005 BC00005
CALL JOB:SEARCH-R1
SET P0097 P0006
SFTON P0097
MOVL C00006 BC00006 V=166.7 PL=0
SFTOF
COMM MOVL C00007 BC00007 V=333.3
MOVL C00008 BC00008 V=333.3
MOVL C00009 BC00009 V=166.7 PL=0
REFP 3 C00010 BC00010
CALL JOB:SEARCH-R1
IMOV P0057 V=23.0
SET P0098 P0006
SFTON P0098
REFP 3 C00011 BC00011
CALL JOB:SEARCH-R1
SET P0098 P0006
SFTON P0098
MOVL C00012 BC00012 V=166.7 PL=0
'TEST
SFTOF
MOVJ C00013 BC00013 VJ=20.00
MOVJ C00014 BC00014 VJ=30.00
'------------------------
'W38 P
'------------------------
'TEST
MOVL C00015 BC00015 V=166.7
MOVL C00016 BC00016 V=166.7 PL=0
REFP 3 C00017 BC00017
CALL JOB:SEARCH-R1
IMOV P0057 V=23.0
SET P0099 P0006
SFTON P0099
REFP 3 C00018 BC00018
CALL JOB:SEARCH-R1
SET P0099 P0006
SFTON P0099
MOVL C00019 BC00019 V=166.7 PL=0
'TEST
SFTOF
MOVL C00020 BC00020 V=333.3
MOVL C00021 BC00021 V=333.3
'------------------------
'W38 L
'------------------------
'TEST
MOVL C00022 BC00022 V=166.7 PL=0
REFP 3 C00023 BC00023
CALL JOB:SEARCH-R1
IMOV P0057 V=23.0
SET P0100 P0006
SFTON P0100
REFP 3 C00024 BC00024
CALL JOB:SEARCH-R1
SET P0100 P0006
SFTON P0100
MOVL C00025 BC00025 V=166.7 PL=0
'TEST
SFTOF
MOVJ C00026 BC00026 VJ=20.00
'------------------------
'W45 P
'------------------------
MOVL C00027 BC00027 V=166.7 PL=0
REFP 3 C00028 BC00028
CALL JOB:SEARCH-R1
IMOV P0057 V=23.0
SET P0101 P0006
SFTON P0101
REFP 3 C00029 BC00029
CALL JOB:SEARCH-R1
SET P0101 P0006
SFTON P0101
MOVL C00030 BC00030 V=166.7 PL=0
'TEST
SFTOF
MOVJ C00031 BC00031 VJ=20.00
'------------------------
'W45 L
'------------------------
MOVL C00032 BC00032 V=133.3 PL=0
REFP 3 C00033 BC00033
CALL JOB:SEARCH-R1
IMOV P0057 V=23.0
SET P0102 P0006
SFTON P0102
REFP 3 C00034 BC00034
CALL JOB:SEARCH-R1
SET P0102 P0006
SFTON P0102
MOVL C00035 BC00035 V=250.0 PL=0
'TEST
SFTOF
MOVJ C00036 BC00036 VJ=20.00
'------------------------
'W48 P
'------------------------
'TEST
MOVL C00037 BC00037 V=133.3 PL=0
REFP 3 C00038 BC00038
CALL JOB:SEARCH-R1
IMOV P0057 V=23.0
SET P0103 P0006
SFTON P0103
REFP 3 C00039 BC00039
CALL JOB:SEARCH-R1
SET P0103 P0006
SFTON P0103
MOVL C00040 BC00040 V=166.7 PL=0
'TEST
SFTOF
MOVJ C00041 BC00041 VJ=30.00
MOVJ C00042 BC00042 VJ=30.00
MOVJ C00043 BC00043 VJ=30.00
MOVJ C00044 BC00044 VJ=30.00
MOVJ C00045 BC00045 VJ=20.00
MOVL C00046 BC00046 V=250.0
'------------------------
'W48 L
'------------------------
SFTOF
MOVL C00047 BC00047 V=133.3 PL=0
REFP 3 C00048 BC00048
CALL JOB:SEARCH-R1
IMOV P0057 V=23.0
SET P0104 P0006
SFTON P0104
REFP 3 C00049 BC00049
CALL JOB:SEARCH-R1
SET P0104 P0006
SFTON P0104
MOVL C00050 BC00050 V=166.7 PL=0
SFTOF
MOVJ C00051 BC00051 VJ=20.00
'------------------------
'W36 P
'------------------------
MOVL C00052 BC00052 V=133.3 PL=0
REFP 3 C00053 BC00053
CALL JOB:SEARCH-R1
IMOV P0057 V=23.0
SET P0105 P0006
SFTON P0105
REFP 3 C00054 BC00054
CALL JOB:SEARCH-R1
SET P0105 P0006
SFTON P0105
MOVL C00055 BC00055 V=166.7 PL=0
'TEST
SFTOF
MOVJ C00056 BC00056 VJ=20.00
'------------------------
'W36 L
'------------------------
MOVL C00057 BC00057 V=166.7 PL=0
REFP 3 C00058 BC00058
CALL JOB:SEARCH-R1
IMOV P0057 V=23.0
SET P0106 P0006
SFTON P0106
REFP 3 C00059 BC00059
CALL JOB:SEARCH-R1
SET P0106 P0006
SFTON P0106
MOVL C00060 BC00060 V=166.7 PL=0
'TEST
MOVJ C00061 BC00061 VJ=20.00
SFTOF
'------------------------
'W44 P
'------------------------
'TEST
MOVL C00062 BC00062 V=133.3 PL=0
REFP 3 C00063 BC00063
CALL JOB:SEARCH-R1
IMOV P0057 V=23.0
SET P0107 P0006
SFTON P0107
REFP 3 C00064 BC00064
CALL JOB:SEARCH-R1
SET P0107 P0006
SFTON P0107
MOVL C00065 BC00065 V=250.0 PL=0
'TEST
SFTOF
MOVL C00066 BC00066 V=250.0
MOVJ C00067 BC00067 VJ=25.00
MOVJ C00068 BC00068 VJ=25.00
MOVJ C00069 BC00069 VJ=25.00
MOVJ C00070 BC00070 VJ=25.00
MOVJ C00071 BC00071 VJ=30.00
MOVJ C00072 BC00072 VJ=25.00
'------------------------
'W44 L
'------------------------
'TEST
MOVL C00073 BC00073 V=166.7 PL=0
REFP 3 C00074 BC00074
CALL JOB:SEARCH-R1
IMOV P0057 V=23.0
SET P0108 P0006
SFTON P0108
REFP 3 C00075 BC00075
CALL JOB:SEARCH-R1
SET P0108 P0006
SFTON P0108
MOVL C00076 BC00076 V=250.0 PL=0
'TEST
SFTOF
MOVL C00077 BC00077 V=250.0
'------------------------
'TEST
MOVL C00078 BC00078 V=166.7 PL=0
REFP 3 C00079 BC00079
CALL JOB:SEARCH-R1
IMOV P0057 V=23.0
SET P0109 P0006
SFTON P0109
REFP 3 C00080 BC00080
CALL JOB:SEARCH-R1
SET P0109 P0006
SFTON P0109
MOVL C00081 BC00081 V=250.0 PL=0
'TEST
SFTOF
'------------------------
'TEST
MOVL C00082 BC00082 V=166.7 PL=0
REFP 3 C00083 BC00083
CALL JOB:SEARCH-R1
IMOV P0057 V=23.0
SET P0110 P0006
SFTON P0110
REFP 3 C00084 BC00084
CALL JOB:SEARCH-R1
SET P0110 P0006
SFTON P0110
MOVL C00085 BC00085 V=250.0 PL=0
'TEST
SFTOF
MOVJ C00086 BC00086 VJ=25.00
CALL JOB:FRONT_SEARCH_0ST-2_5240_V2
COMM MOVJ C00087 BC00087 VJ=20.00
COMM MOVJ C00088 BC00088 VJ=20.00
COMM MOVJ C00089 BC00089 VJ=20.00
COMM 'DODANE
COMM 'SZUKANIE FRONT
COMM '------------------------
COMM '503
COMM '------------------------
COMM MOVL C00090 BC00090 V=333.3
COMM MOVL C00091 BC00091 V=166.7 PL=0
COMM REFP 3 C00092 BC00092
COMM CALL JOB:SEARCH-R1
COMM IMOV P0058 V=16.7
COMM SET P0350 P0006
COMM SFTON P0350
COMM REFP 3 C00093 BC00093
COMM CALL JOB:SEARCH-R1
COMM SET P0350 P0006
COMM SFTON P0350
COMM MOVL C00094 BC00094 V=66.7 PL=0
COMM SFTOF
COMM '------------------------
COMM '------------------------
COMM '502
COMM '------------------------
COMM MOVL C00095 BC00095 V=166.7
COMM MOVL C00096 BC00096 V=66.7 PL=0
COMM REFP 3 C00097 BC00097
COMM CALL JOB:SEARCH-R1
COMM IMOV P0058 V=16.7
COMM SET P0351 P0006
COMM SFTON P0351
COMM REFP 3 C00098 BC00098
COMM CALL JOB:SEARCH-R1
COMM SET P0351 P0006
COMM SFTON P0351
COMM MOVL C00099 BC00099 V=66.7 PL=0
COMM SFTOF
COMM '------------------------
COMM '------------------------
COMM '501
COMM '------------------------
COMM MOVL C00100 BC00100 V=166.7
COMM MOVL C00101 BC00101 V=66.7 PL=0
COMM REFP 3 C00102 BC00102
COMM CALL JOB:SEARCH-R1
COMM IMOV P0058 V=16.7
COMM SET P0352 P0006
COMM SFTON P0352
COMM REFP 3 C00103 BC00103
COMM CALL JOB:SEARCH-R1
COMM SET P0352 P0006
COMM SFTON P0352
COMM MOVL C00104 BC00104 V=66.7 PL=0
COMM SFTOF
COMM '------------------------
COMM '------------------------
COMM '500
COMM '------------------------
COMM MOVL C00105 BC00105 V=166.7
COMM MOVL C00106 BC00106 V=66.7 PL=0
COMM REFP 3 C00107 BC00107
COMM CALL JOB:SEARCH-R1
COMM IMOV P0058 V=16.7
COMM SET P0353 P0006
COMM SFTON P0353
COMM REFP 3 C00108 BC00108
COMM CALL JOB:SEARCH-R1
COMM SET P0353 P0006
COMM SFTON P0353
COMM MOVL C00109 BC00109 V=66.7 PL=0
COMM SFTOF
COMM '------------------------
COMM MOVL C00110 BC00110 V=333.3
COMM MOVL C00111 BC00111 V=333.3
COMM MOVJ C00112 BC00112 VJ=10.00
COMM 'DODANE
COMM MOVJ C00113 BC00113 VJ=10.00
COMM '------------------------
COMM 'SFT402
COMM '------------------------
COMM SFTOF
COMM MOVL C00114 BC00114 V=150.0
COMM MOVL C00115 BC00115 V=66.7 PL=0
COMM REFP 3 C00116 BC00116
COMM CALL JOB:SEARCH-R1
COMM SET P0402 P0006
COMM SFTON P0402
COMM MOVL C00117 BC00117 V=150.0
COMM MOVL C00118 BC00118 V=66.7 PL=0
COMM REFP 3 C00119 BC00119
COMM CALL JOB:SEARCH-R1
COMM SET P0402 P0006
COMM SFTON P0402
COMM MOVL C00120 BC00120 V=133.3
COMM MOVL C00121 BC00121 V=150.0
COMM MOVL C00122 BC00122 V=150.0
COMM MOVL C00123 BC00123 V=66.7 PL=0
COMM REFP 3 C00124 BC00124
COMM CALL JOB:SEARCH-R1
COMM SET P0402 P0006
COMM SFTOF
COMM MOVL C00125 BC00125 V=150.0
COMM '------------------------
COMM 'SFT403
COMM '------------------------
COMM 'START
COMM SFTOF
COMM MOVL C00126 BC00126 V=250.0
COMM MOVL C00127 BC00127 V=133.3 PL=0
COMM REFP 3 C00128 BC00128
COMM CALL JOB:SEARCH-R1
COMM SET P0416 P0006
COMM SFTON P0416
COMM MOVL C00129 BC00129 V=133.3
COMM REFP 3 C00130 BC00130
COMM CALL JOB:SEARCH-R1
COMM SET P0402 P0006
COMM SFTOF
COMM MOVL C00131 BC00131 V=150.0
COMM '------------------------
COMM '------------------------
COMM SFTOF
COMM MOVL C00132 BC00132 V=250.0
COMM MOVL C00133 BC00133 V=133.3 PL=0
COMM REFP 3 C00134 BC00134
COMM CALL JOB:SEARCH-R1
COMM SET P0403 P0006
COMM SFTON P0403
COMM MOVL C00135 BC00135 V=66.7 PL=0
COMM REFP 3 C00136 BC00136
COMM CALL JOB:SEARCH-R1
COMM SET P0403 P0006
COMM SFTOF
COMM MOVL C00137 BC00137 V=150.0
COMM MOVJ C00138 BC00138 VJ=20.00
COMM MOVJ C00139 BC00139 VJ=20.00
COMM '------------------------
COMM 'SFT401
COMM '------------------------
COMM SFTOF
COMM MOVL C00140 BC00140 V=150.0
COMM MOVL C00141 BC00141 V=66.7 PL=0
COMM REFP 3 C00142 BC00142
COMM CALL JOB:SEARCH-R1
COMM SET P0401 P0006
COMM SFTON P0401
COMM MOVL C00143 BC00143 V=66.7 PL=0
COMM REFP 3 C00144 BC00144
COMM CALL JOB:SEARCH-R1
COMM SET P0401 P0006
COMM SFTOF
COMM MOVL C00145 BC00145 V=150.0
COMM 'SFT400
COMM '------------------------
COMM SFTOF
COMM MOVL C00146 BC00146 V=333.3
COMM MOVL C00147 BC00147 V=66.7 PL=0
COMM REFP 3 C00148 BC00148
COMM CALL JOB:SEARCH-R1
COMM SET P0405 P0006
COMM SFTON P0405
COMM MOVL C00149 BC00149 V=66.7 PL=0
COMM REFP 3 C00150 BC00150
COMM CALL JOB:SEARCH-R1
COMM SET P0405 P0006
COMM SFTOF
COMM MOVL C00151 BC00151 V=150.0
COMM 'SFT400
COMM '------------------------
COMM SFTOF
COMM MOVL C00152 BC00152 V=333.3
COMM MOVL C00153 BC00153 V=133.3 PL=0
COMM REFP 3 C00154 BC00154
COMM CALL JOB:SEARCH-R1
COMM SET P0406 P0006
COMM SFTON P0406
COMM MOVL C00155 BC00155 V=66.7 PL=0
COMM REFP 3 C00156 BC00156
COMM CALL JOB:SEARCH-R1
COMM SET P0406 P0006
COMM SFTOF
COMM MOVL C00157 BC00157 V=150.0
COMM 'SFT400
COMM '------------------------
COMM SFTOF
COMM MOVL C00158 BC00158 V=150.0
COMM MOVL C00159 BC00159 V=66.7 PL=0
COMM REFP 3 C00160 BC00160
COMM CALL JOB:SEARCH-R1
COMM SET P0400 P0006
COMM SFTON P0400
COMM MOVL C00161 BC00161 V=150.0
COMM MOVL C00162 BC00162 V=66.7 PL=0
COMM REFP 3 C00163 BC00163
COMM CALL JOB:SEARCH-R1
COMM SET P0400 P0006
COMM SFTON P0400
COMM MOVL C00164 BC00164 V=150.0
COMM MOVL C00165 BC00165 V=150.0
COMM MOVL C00166 BC00166 V=66.7 PL=0
COMM REFP 3 C00167 BC00167
COMM CALL JOB:SEARCH-R1
COMM SET P0400 P0006
COMM SFTOF
COMM MOVL C00168 BC00168 V=83.3
COMM MOVL C00169 BC00169 V=250.0
COMM MOVL C00170 BC00170 V=333.3
COMM MOVL C00171 BC00171 V=66.7 PL=0
COMM REFP 3 C00172 BC00172
COMM CALL JOB:SEARCH-R1
COMM SET P0415 P0006
COMM SFTON P0415
COMM MOVL C00173 BC00173 V=133.3
COMM REFP 3 C00174 BC00174
COMM CALL JOB:SEARCH-R1
COMM SET P0415 P0006
COMM SFTOF
COMM MOVL C00175 BC00175 V=150.0
COMM '------------------------
COMM 'SFT403
COMM '------------------------
COMM 'START
COMM SFTOF
COMM MOVJ C00176 BC00176 VJ=10.00
COMM '------------------------
COMM 'SFT399
COMM '------------------------
COMM 'START
COMM SFTOF
COMM MOVL C00177 BC00177 V=150.0
COMM MOVL C00178 BC00178 V=66.7 PL=0
COMM REFP 3 C00179 BC00179
COMM CALL JOB:SEARCH-R1
COMM SET P0399 P0006
COMM SFTON P0399
COMM MOVL C00180 BC00180 V=66.7 PL=0
COMM REFP 3 C00181 BC00181
COMM CALL JOB:SEARCH-R1
COMM SET P0399 P0006
COMM SFTOF
COMM MOVL C00182 BC00182 V=150.0
COMM MOVJ C00183 BC00183 VJ=20.00
COMM MOVJ C00184 BC00184 VJ=30.00
MOVJ C00185 BC00185 VJ=30.00
MOVJ C00186 BC00186 VJ=30.00
MOVJ C00187 BC00187 VJ=40.00
'WELD
'WELD
MOVJ C00188 BC00188 VJ=20.00
'**********************
'W36
'**********************
MOVL C00189 BC00189 V=500.0
SFTON P0105
MOVL C00190 BC00190 V=166.7 PL=0
SFTOF
MACRO1 MJ#(0) ARGF24
ARCON
SFTON P0106
MOVL C00191 BC00191 V=11.7
ARCOF
SFTOF
MOVJ C00192 BC00192 VJ=15.00
MOVJ C00193 BC00193 VJ=10.00
MOVJ C00194 BC00194 VJ=10.00
MOVJ C00195 BC00195 VJ=10.00
MOVJ C00196 BC00196 VJ=30.00
MOVJ C00197 BC00197 VJ=20.00
MOVJ C00198 BC00198 VJ=10.00
MOVJ C00199 BC00199 VJ=15.00
'**********************
'W38
'**********************
MOVL C00200 BC00200 V=500.0
SFTON P0100
MOVL C00201 BC00201 V=166.7 PL=0
SFTOF
ARCON
SFTON P0099
MOVL C00202 BC00202 V=11.3
ARCOF
SFTOF
'DODANE
MOVL C00203 BC00203 V=500.0
MOVJ C00204 BC00204 VJ=10.00
MOVJ C00205 BC00205 VJ=10.00
MOVJ C00206 BC00206 VJ=10.00
MOVJ C00207 BC00207 VJ=10.00
MOVJ C00208 BC00208 VJ=25.00
MOVJ C00209 BC00209 VJ=30.00
MOVJ C00210 BC00210 VJ=30.00
MOVJ C00211 BC00211 VJ=30.00
MOVL C00212 BC00212 V=500.0
SFTON P0107
MOVL C00213 BC00213 V=166.7 PL=0
SFTOF
MACRO1 MJ#(0) ARGF24
ARCON
SFTON P0108
MOVL C00214 BC00214 V=10.8
MOVL C00215 BC00215 V=10.8
ARCOF
SFTOF
MOVL C00216 BC00216 V=500.0
MOVL C00217 BC00217 V=500.0
MOVJ C00218 BC00218 VJ=10.00
MOVJ C00219 BC00219 VJ=10.00
MOVJ C00220 BC00220 VJ=20.00
'**********************
'DODATEK
'**********************
MOVJ C00221 BC00221 VJ=10.00
MOVJ C00222 BC00222 VJ=10.00
MOVJ C00223 BC00223 VJ=20.00
MOVJ C00224 BC00224 VJ=20.00
MOVJ C00225 BC00225 VJ=20.00
MOVL C00226 BC00226 V=333.3
MOVL C00227 BC00227 V=166.7
MACRO1 MJ#(0) ARGF24
SFTON P0109
MOVL C00228 BC00228 V=166.7 PL=0
SFTOF
ARCON
SFTON P0110
MOVL C00229 BC00229 V=10.8
ARCOF
SFTOF
MOVL C00230 BC00230 V=500.0
MOVJ C00231 BC00231 VJ=20.00
MOVJ C00232 BC00232 VJ=30.00
'**********************
'W45
'**********************
MOVJ C00233 BC00233 VJ=30.00
MOVJ C00234 BC00234 VJ=20.00
MOVJ C00235 BC00235 VJ=10.00
MACRO1 MJ#(0) ARGF24
MOVL C00236 BC00236 V=500.0
SFTON P0102
MOVL C00237 BC00237 V=166.7 PL=0
SFTOF
ARCON
SFTON P0101
MOVL C00238 BC00238 V=11.7
ARCOF
SFTOF
MOVL C00239 BC00239 V=500.0
'**********************
'SPOINA_PODLOGA_BRAK_ROZP
'**********************
MOVL C00240 BC00240 V=500.0
MOVL C00241 BC00241 V=500.0
SFTON P0098
MOVL C00242 BC00242 V=166.7 PL=0
SFTOF
ARCON
SFTON P0097
MOVL C00243 BC00243 V=11.3
ARCOF
SFTOF
'DODANE
MOVL C00244 BC00244 V=500.0
MOVJ C00245 BC00245 VJ=10.00
MOVJ C00246 BC00246 VJ=10.00
'**********************
'W48
'**********************
MOVJ C00247 BC00247 VJ=15.00
MOVJ C00248 BC00248 VJ=15.00
MOVJ C00249 BC00249 VJ=15.00
SFTON P0103
MOVL C00250 BC00250 V=166.7 PL=0
ARCON
SFTON P0104
MOVL C00251 BC00251 V=10.8
ARCOF
SFTOF
MOVL C00252 BC00252 V=500.0
MOVJ C00253 BC00253 VJ=15.00
MOVJ C00254 BC00254 VJ=20.00
MOVJ C00255 BC00255 VJ=40.00
CALL JOB:FRONT_WELD_0ST-2_5240_V2
CALL JOB:MOVE_OUT_OF_TUNNEL
CALL JOB:CLEAN-R1
CALL JOB:MOVE_INTO_TUNNEL
MOVJ C00256 BC00256 VJ=30.00 PL=0
'------------------------
'------------------------
'PRAWA STRONA PROFIL GORA
'------------------------
'------------------------
MOVJ C00257 BC00257 VJ=20.00
'------------------------
'W51A L
'------------------------
SFTOF
MOVJ C00258 BC00258 VJ=10.00
MOVL C00259 BC00259 V=66.7 PL=0
REFP 3 C00260 BC00260
CALL JOB:SEARCH-R1
SET P0299 P0006
SFTON P0299
MOVL C00261 BC00261 V=66.7 PL=0
REFP 3 C00262 BC00262
CALL JOB:SEARCH-R1
SET P0299 P0006
SFTON P0299
MOVL C00263 BC00263 V=83.3
MOVL C00264 BC00264 V=166.7 PL=0
REFP 3 C00265 BC00265
CALL JOB:SEARCH-R1
SET P0299 P0006
SFTON P0299
MOVL C00266 BC00266 V=133.3 PL=0
SFTOF
'------------------------
'W51A P
'------------------------
SFTOF
MOVL C00267 BC00267 V=250.0
MOVL C00268 BC00268 V=66.7 PL=0
REFP 3 C00269 BC00269
CALL JOB:SEARCH-R1
SET P0300 P0006
SFTON P0300
MOVL C00270 BC00270 V=66.7 PL=0
REFP 3 C00271 BC00271
CALL JOB:SEARCH-R1
SET P0300 P0006
SFTON P0300
MOVL C00272 BC00272 V=66.7 PL=0
SFTOF
'------------------------
'W54A L
'------------------------
SFTOF
MOVJ C00273 BC00273 VJ=30.00
MOVL C00274 BC00274 V=133.3 PL=0
REFP 3 C00275 BC00275
CALL JOB:SEARCH-R1
SET P0301 P0006
SFTON P0301
MOVL C00276 BC00276 V=66.7 PL=0
REFP 3 C00277 BC00277
CALL JOB:SEARCH-R1
SET P0301 P0006
SFTON P0301
MOVL C00278 BC00278 V=66.7 PL=0
SFTOF
'------------------------
'W54A P
'------------------------
SFTOF
MOVJ C00279 BC00279 VJ=30.00
MOVL C00280 BC00280 V=133.3 PL=0
REFP 3 C00281 BC00281
CALL JOB:SEARCH-R1
SET P0302 P0006
SFTON P0302
MOVL C00282 BC00282 V=66.7 PL=0
REFP 3 C00283 BC00283
CALL JOB:SEARCH-R1
SET P0302 P0006
SFTON P0302
MOVL C00284 BC00284 V=66.7 PL=0
SFTOF
'------------------------
'W50A L
'------------------------
SFTOF
MOVJ C00285 BC00285 VJ=30.00
MOVL C00286 BC00286 V=133.3 PL=0
REFP 3 C00287 BC00287
CALL JOB:SEARCH-R1
SET P0303 P0006
SFTON P0303
MOVL C00288 BC00288 V=66.7 PL=0
REFP 3 C00289 BC00289
CALL JOB:SEARCH-R1
SET P0303 P0006
SFTON P0303
MOVL C00290 BC00290 V=66.7 PL=0
SFTOF
'------------------------
'W50A P
'------------------------
SFTOF
MOVJ C00291 BC00291 VJ=30.00
MOVL C00292 BC00292 V=133.3 PL=0
REFP 3 C00293 BC00293
CALL JOB:SEARCH-R1
SET P0304 P0006
SFTON P0304
MOVL C00294 BC00294 V=66.7 PL=0
REFP 3 C00295 BC00295
CALL JOB:SEARCH-R1
SET P0304 P0006
SFTON P0304
MOVL C00296 BC00296 V=66.7 PL=0
SFTOF
'------------------------
'W53A L
'------------------------
SFTOF
MOVJ C00297 BC00297 VJ=30.00
MOVL C00298 BC00298 V=133.3 PL=0
REFP 3 C00299 BC00299
CALL JOB:SEARCH-R1
SET P0305 P0006
SFTON P0305
MOVL C00300 BC00300 V=66.7 PL=0
REFP 3 C00301 BC00301
CALL JOB:SEARCH-R1
SET P0305 P0006
SFTON P0305
MOVL C00302 BC00302 V=66.7 PL=0
SFTOF
'------------------------
'W53A P
'------------------------
SFTOF
MOVJ C00303 BC00303 VJ=30.00
MOVL C00304 BC00304 V=200.0
MOVL C00305 BC00305 V=66.7 PL=0
REFP 3 C00306 BC00306
CALL JOB:SEARCH-R1
SET P0306 P0006
SFTON P0306
MOVL C00307 BC00307 V=66.7 PL=0
REFP 3 C00308 BC00308
CALL JOB:SEARCH-R1
SET P0306 P0006
SFTON P0306
MOVL C00309 BC00309 V=66.7 PL=0
SFTOF
'------------------------
'W56A L
'------------------------
SFTOF
MOVJ C00310 BC00310 VJ=30.00
MOVL C00311 BC00311 V=133.3 PL=0
REFP 3 C00312 BC00312
CALL JOB:SEARCH-R1
SET P0307 P0006
SFTON P0307
MOVL C00313 BC00313 V=66.7 PL=0
REFP 3 C00314 BC00314
CALL JOB:SEARCH-R1
SET P0307 P0006
SFTON P0307
MOVL C00315 BC00315 V=66.7 PL=0
SFTOF
'------------------------
'W56A P
'------------------------
SFTOF
MOVJ C00316 BC00316 VJ=30.00
MOVL C00317 BC00317 V=133.3 PL=0
REFP 3 C00318 BC00318
CALL JOB:SEARCH-R1
SET P0308 P0006
SFTON P0308
MOVL C00319 BC00319 V=66.7 PL=0
REFP 3 C00320 BC00320
CALL JOB:SEARCH-R1
SET P0308 P0006
SFTON P0308
MOVL C00321 BC00321 V=66.7 PL=0
SFTOF
'------------------------
'W52A L
'------------------------
SFTOF
MOVJ C00322 BC00322 VJ=30.00
MOVL C00323 BC00323 V=250.0
MOVL C00324 BC00324 V=66.7 PL=0
REFP 3 C00325 BC00325
CALL JOB:SEARCH-R1
SET P0309 P0006
SFTON P0309
MOVL C00326 BC00326 V=66.7 PL=0
REFP 3 C00327 BC00327
CALL JOB:SEARCH-R1
SET P0309 P0006
SFTON P0309
MOVL C00328 BC00328 V=66.7 PL=0
SFTOF
'------------------------
'W52A P
'------------------------
SFTOF
MOVJ C00329 BC00329 VJ=5.00
MOVJ C00330 BC00330 VJ=20.00
MOVL C00331 BC00331 V=116.7 PL=0
REFP 3 C00332 BC00332
CALL JOB:SEARCH-R1
SET P0310 P0006
SFTON P0310
MOVL C00333 BC00333 V=66.7 PL=0
REFP 3 C00334 BC00334
CALL JOB:SEARCH-R1
SET P0310 P0006
SFTON P0310
MOVL C00335 BC00335 V=66.7 PL=0
SFTOF
'------------------------
'W55A L
'------------------------
SFTOF
MOVL C00336 BC00336 V=250.0
MOVJ C00337 BC00337 VJ=10.00
MOVL C00338 BC00338 V=66.7 PL=0
REFP 3 C00339 BC00339
CALL JOB:SEARCH-R1
SET P0311 P0006
SFTON P0311
MOVL C00340 BC00340 V=66.7 PL=0
REFP 3 C00341 BC00341
CALL JOB:SEARCH-R1
SET P0311 P0006
SFTON P0311
MOVL C00342 BC00342 V=66.7 PL=0
SFTOF
'------------------------
'W55A P
'------------------------
SFTOF
MOVL C00343 BC00343 V=250.0
MOVL C00344 BC00344 V=166.7
MOVL C00345 BC00345 V=66.7 PL=0
REFP 3 C00346 BC00346
CALL JOB:SEARCH-R1
SET P0312 P0006
SFTON P0312
MOVL C00347 BC00347 V=66.7 PL=0
REFP 3 C00348 BC00348
CALL JOB:SEARCH-R1
SET P0312 P0006
SFTON P0312
MOVL C00349 BC00349 V=66.7 PL=0
MOVL C00350 BC00350 V=166.7
SFTOF
MOVL C00351 BC00351 V=250.0
MOVJ C00352 BC00352 VJ=20.00
MOVJ C00353 BC00353 VJ=20.00
MOVJ C00354 BC00354 VJ=20.00
MOVJ C00355 BC00355 VJ=20.00
MOVJ C00356 BC00356 VJ=20.00
MOVJ C00357 BC00357 VJ=20.00
'------------------------
'------------------------
'LEWA STRONA PROFIL GORA
'------------------------
'------------------------
MOVJ C00358 BC00358 VJ=10.00
'------------------------
'W55B L
'------------------------
SFTOF
MOVJ C00359 BC00359 VJ=10.00
MOVL C00360 BC00360 V=66.7 PL=0
REFP 3 C00361 BC00361
CALL JOB:SEARCH-R1
SET P0349 P0006
SFTON P0349
MOVL C00362 BC00362 V=66.7 PL=0
REFP 3 C00363 BC00363
CALL JOB:SEARCH-R1
SET P0349 P0006
SFTON P0349
MOVL C00364 BC00364 V=66.7 PL=0
SFTOF
MOVJ C00365 BC00365 VJ=10.00
MOVJ C00366 BC00366 VJ=10.00
'------------------------
'W55B P
'------------------------
SFTOF
MOVL C00367 BC00367 V=66.7 PL=0
REFP 3 C00368 BC00368
CALL JOB:SEARCH-R1
SET P0350 P0006
SFTON P0350
MOVL C00369 BC00369 V=66.7 PL=0
REFP 3 C00370 BC00370
CALL JOB:SEARCH-R1
SET P0350 P0006
SFTON P0350
MOVL C00371 BC00371 V=66.7 PL=0
SFTOF
'------------------------
'W52B L
'------------------------
SFTOF
MOVJ C00372 BC00372 VJ=20.00
MOVJ C00373 BC00373 VJ=20.00
MOVL C00374 BC00374 V=150.0
MOVL C00375 BC00375 V=66.7 PL=0
REFP 3 C00376 BC00376
CALL JOB:SEARCH-R1
SET P0351 P0006
SFTON P0351
MOVL C00377 BC00377 V=66.7 PL=0
REFP 3 C00378 BC00378
CALL JOB:SEARCH-R1
SET P0351 P0006
SFTON P0351
MOVL C00379 BC00379 V=66.7 PL=0
SFTOF
'------------------------
'W52B P
'------------------------
SFTOF
MOVJ C00380 BC00380 VJ=30.00
MOVL C00381 BC00381 V=116.7 PL=0
REFP 3 C00382 BC00382
CALL JOB:SEARCH-R1
SET P0352 P0006
SFTON P0352
MOVL C00383 BC00383 V=66.7 PL=0
REFP 3 C00384 BC00384
CALL JOB:SEARCH-R1
SET P0352 P0006
SFTON P0352
MOVL C00385 BC00385 V=66.7 PL=0
SFTOF
'------------------------
'W56B L
'------------------------
SFTOF
MOVJ C00386 BC00386 VJ=30.00
MOVL C00387 BC00387 V=116.7 PL=0
REFP 3 C00388 BC00388
CALL JOB:SEARCH-R1
SET P0353 P0006
SFTON P0353
MOVL C00389 BC00389 V=66.7 PL=0
REFP 3 C00390 BC00390
CALL JOB:SEARCH-R1
SET P0353 P0006
SFTON P0353
MOVL C00391 BC00391 V=66.7 PL=0
SFTOF
'------------------------
'W56B P
'------------------------
SFTOF
MOVJ C00392 BC00392 VJ=30.00
MOVL C00393 BC00393 V=116.7 PL=0
REFP 3 C00394 BC00394
CALL JOB:SEARCH-R1
SET P0354 P0006
SFTON P0354
MOVL C00395 BC00395 V=66.7 PL=0
REFP 3 C00396 BC00396
CALL JOB:SEARCH-R1
SET P0354 P0006
SFTON P0354
MOVL C00397 BC00397 V=66.7 PL=0
SFTOF
'------------------------
'W53B L
'------------------------
SFTOF
MOVJ C00398 BC00398 VJ=30.00
MOVL C00399 BC00399 V=116.7 PL=0
REFP 3 C00400 BC00400
CALL JOB:SEARCH-R1
SET P0355 P0006
SFTON P0355
MOVL C00401 BC00401 V=66.7 PL=0
REFP 3 C00402 BC00402
CALL JOB:SEARCH-R1
SET P0355 P0006
SFTON P0355
MOVL C00403 BC00403 V=66.7 PL=0
SFTOF
'------------------------
'W53B P
'------------------------
SFTOF
MOVJ C00404 BC00404 VJ=30.00
MOVL C00405 BC00405 V=116.7 PL=0
REFP 3 C00406 BC00406
CALL JOB:SEARCH-R1
SET P0356 P0006
SFTON P0356
MOVL C00407 BC00407 V=66.7 PL=0
REFP 3 C00408 BC00408
CALL JOB:SEARCH-R1
SET P0356 P0006
SFTON P0356
MOVL C00409 BC00409 V=66.7 PL=0
SFTOF
'------------------------
'W50B L
'------------------------
SFTOF
MOVJ C00410 BC00410 VJ=30.00
MOVL C00411 BC00411 V=116.7 PL=0
REFP 3 C00412 BC00412
CALL JOB:SEARCH-R1
SET P0357 P0006
SFTON P0357
MOVL C00413 BC00413 V=66.7 PL=0
REFP 3 C00414 BC00414
CALL JOB:SEARCH-R1
SET P0357 P0006
SFTON P0357
MOVL C00415 BC00415 V=66.7 PL=0
SFTOF
'------------------------
'W50B P
'------------------------
SFTOF
MOVJ C00416 BC00416 VJ=30.00
MOVL C00417 BC00417 V=116.7 PL=0
REFP 3 C00418 BC00418
CALL JOB:SEARCH-R1
SET P0358 P0006
SFTON P0358
MOVL C00419 BC00419 V=66.7 PL=0
REFP 3 C00420 BC00420
CALL JOB:SEARCH-R1
SET P0358 P0006
SFTON P0358
MOVL C00421 BC00421 V=66.7 PL=0
SFTOF
'------------------------
'W54B L
'------------------------
SFTOF
MOVJ C00422 BC00422 VJ=30.00
MOVL C00423 BC00423 V=116.7 PL=0
REFP 3 C00424 BC00424
CALL JOB:SEARCH-R1
SET P0359 P0006
SFTON P0359
MOVL C00425 BC00425 V=66.7 PL=0
REFP 3 C00426 BC00426
CALL JOB:SEARCH-R1
SET P0359 P0006
SFTON P0359
MOVL C00427 BC00427 V=66.7 PL=0
SFTOF
'------------------------
'W54B P
'------------------------
SFTOF
MOVJ C00428 BC00428 VJ=30.00
MOVL C00429 BC00429 V=116.7 PL=0
REFP 3 C00430 BC00430
CALL JOB:SEARCH-R1
SET P0360 P0006
SFTON P0360
MOVL C00431 BC00431 V=66.7 PL=0
REFP 3 C00432 BC00432
CALL JOB:SEARCH-R1
SET P0360 P0006
SFTON P0360
MOVL C00433 BC00433 V=66.7 PL=0
SFTOF
'------------------------
'W51B L
'------------------------
SFTOF
MOVJ C00434 BC00434 VJ=30.00
MOVL C00435 BC00435 V=133.3 PL=0
REFP 3 C00436 BC00436
CALL JOB:SEARCH-R1
SET P0361 P0006
SFTON P0361
MOVL C00437 BC00437 V=66.7 PL=0
REFP 3 C00438 BC00438
CALL JOB:SEARCH-R1
SET P0361 P0006
SFTON P0361
MOVL C00439 BC00439 V=66.7 PL=0
SFTOF
'------------------------
'W51B P
'------------------------
SFTOF
MOVL C00440 BC00440 V=150.0
MOVL C00441 BC00441 V=66.7 PL=0
REFP 3 C00442 BC00442
CALL JOB:SEARCH-R1
SET P0361 P0006
SFTON P0361
MOVL C00443 BC00443 V=66.7 PL=0
REFP 3 C00444 BC00444
CALL JOB:SEARCH-R1
SET P0361 P0006
SFTON P0361
MOVL C00445 BC00445 V=83.3
MOVL C00446 BC00446 V=133.3 PL=0
REFP 3 C00447 BC00447
CALL JOB:SEARCH-R1
SET P0361 P0006
SFTON P0361
SFTOF
MOVL C00448 BC00448 V=83.3
MOVJ C00449 BC00449 VJ=20.00
MOVJ C00450 BC00450 VJ=30.00
MOVJ C00451 BC00451 VJ=10.00
MOVJ C00452 BC00452 VJ=40.00
'**********************
'**********************
'POCZATEK SPAWANIA BOKI
'**********************
'**********************
MOVJ C00453 BC00453 VJ=30.00
MOVJ C00454 BC00454 VJ=20.00
'**********************
'W50A
'**********************
MOVL C00455 BC00455 V=250.0
SFTON P0304
MOVL C00456 BC00456 V=83.3 PL=0
SFTOF
MACRO1 MJ#(0) ARGF10
ARCON
SFTON P0303
MOVL C00457 BC00457 V=10.8
ARCOF
SFTOF
MOVL C00458 BC00458 V=250.0
'W13B
MOVJ C00459 BC00459 VJ=20.00
MOVJ C00460 BC00460 VJ=40.00
MOVJ C00461 BC00461 VJ=20.00
MOVJ C00462 BC00462 VJ=20.00
MOVJ C00463 BC00463 VJ=20.00
'**********************
'W50B
'**********************
MOVL C00464 BC00464 V=250.0
SFTON P0357
MOVL C00465 BC00465 V=166.7 PL=0
SFTOF
MACRO1 MJ#(0) ARGF10
ARCON
SFTON P0358
MOVL C00466 BC00466 V=10.8
ARCOF
SFTOF
MOVL C00467 BC00467 V=250.0
MOVJ C00468 BC00468 VJ=20.00
MOVJ C00469 BC00469 VJ=20.00
MOVJ C00470 BC00470 VJ=20.00
MOVJ C00471 BC00471 VJ=20.00
'**********************
'W51A
'**********************
MOVL C00472 BC00472 V=416.7
MOVL C00473 BC00473 V=416.7
SFTON P0300
MOVL C00474 BC00474 V=166.7 PL=0
SFTOF
MACRO1 MJ#(0) ARGF10
ARCON
SFTON P0299
MOVL C00475 BC00475 V=10.8
MOVL C00476 BC00476 V=10.8
ARCOF
MOVL C00477 BC00477 V=166.7
MOVL C00478 BC00478 V=133.3 PL=0
ARCON
MOVL C00479 BC00479 V=8.3
ARCOF
SFTOF
MOVL C00480 BC00480 V=200.0
MOVJ C00481 BC00481 VJ=30.00
MOVJ C00482 BC00482 VJ=30.00
MOVJ C00483 BC00483 VJ=30.00
MOVJ C00484 BC00484 VJ=30.00
MOVJ C00485 BC00485 VJ=30.00
'**********************
'W51B
'**********************
MOVL C00486 BC00486 V=416.7
MOVL C00487 BC00487 V=416.7
SFTON P0361
MOVL C00488 BC00488 V=166.7 PL=0
SFTOF
MACRO1 MJ#(0) ARGF10
ARCON
SFTON P0362
MOVL C00489 BC00489 V=10.8
MOVL C00490 BC00490 V=10.8
ARCOF
MOVL C00491 BC00491 V=166.7
MACRO1 MJ#(0) ARGF9
MOVL C00492 BC00492 V=166.7 PL=0
ARCON
MOVL C00493 BC00493 V=8.3
ARCOF
SFTOF
MOVL C00494 BC00494 V=166.7
MOVL C00495 BC00495 V=250.0
MOVJ C00496 BC00496 VJ=30.00
MOVJ C00497 BC00497 VJ=30.00
MOVJ C00498 BC00498 VJ=30.00
MOVJ C00499 BC00499 VJ=40.00
MOVJ C00500 BC00500 VJ=40.00
MOVJ C00501 BC00501 VJ=20.00
MOVJ C00502 BC00502 VJ=20.00
MOVJ C00503 BC00503 VJ=20.00
MOVJ C00504 BC00504 VJ=20.00
MOVJ C00505 BC00505 VJ=20.00
'**********************
'W52A
'**********************
SFTON P0310
MOVL C00506 BC00506 V=250.0
MOVL C00507 BC00507 V=83.3 PL=0
SFTOF
MACRO1 MJ#(0) ARGF10
ARCON
SFTON P0309
MOVL C00508 BC00508 V=10.8
ARCOF
SFTOF
MOVL C00509 BC00509 V=333.3
MOVJ C00510 BC00510 VJ=30.00
MOVJ C00511 BC00511 VJ=30.00
MOVJ C00512 BC00512 VJ=30.00
MOVJ C00513 BC00513 VJ=30.00
MOVJ C00514 BC00514 VJ=30.00
MOVJ C00515 BC00515 VJ=20.00
MOVJ C00516 BC00516 VJ=20.00
MOVJ C00517 BC00517 VJ=20.00
'**********************
'52B
'**********************
MOVL C00518 BC00518 V=250.0
SFTON P0351
MOVL C00519 BC00519 V=83.3 PL=0
SFTOF
MACRO1 MJ#(0) ARGF10
ARCON
SFTON P0352
MOVL C00520 BC00520 V=10.8
ARCOF
MOVL C00521 BC00521 V=333.3
SFTOF
MOVJ C00522 BC00522 VJ=20.00
MOVJ C00523 BC00523 VJ=30.00
MOVJ C00524 BC00524 VJ=30.00
'**********************
'W53A
'**********************
MOVJ C00525 BC00525 VJ=30.00
MOVJ C00526 BC00526 VJ=30.00
MOVJ C00527 BC00527 VJ=10.00
'**********************
'W53A
'**********************
SFTON P0306
MOVL C00528 BC00528 V=250.0
MOVL C00529 BC00529 V=83.3 PL=0
SFTOF
MACRO1 MJ#(0) ARGF10
ARCON
SFTON P0305
MOVL C00530 BC00530 V=10.8
ARCOF
SFTOF
MOVL C00531 BC00531 V=250.0
MOVJ C00532 BC00532 VJ=30.00
MOVJ C00533 BC00533 VJ=30.00
MOVJ C00534 BC00534 VJ=30.00
MOVJ C00535 BC00535 VJ=30.00
MOVJ C00536 BC00536 VJ=30.00
MOVJ C00537 BC00537 VJ=30.00
MOVL C00538 BC00538 V=250.0
'**********************
'W53B
'**********************
SFTON P0355
MOVL C00539 BC00539 V=250.0
MOVL C00540 BC00540 V=83.3 PL=0
SFTOF
MACRO1 MJ#(0) ARGF10
ARCON
SFTON P0356
MOVL C00541 BC00541 V=10.8
ARCOF
SFTOF
MOVL C00542 BC00542 V=333.3
MOVJ C00543 BC00543 VJ=30.00
MOVJ C00544 BC00544 VJ=30.00
MOVJ C00545 BC00545 VJ=30.00
MOVJ C00546 BC00546 VJ=30.00
MOVJ C00547 BC00547 VJ=30.00
'**********************
'W54A
'**********************
SFTON P0302
MOVL C00548 BC00548 V=250.0
MOVL C00549 BC00549 V=83.3 PL=0
SFTOF
MACRO1 MJ#(0) ARGF10
ARCON
SFTON P0301
MOVL C00550 BC00550 V=10.8
ARCOF
SFTOF
MOVL C00551 BC00551 V=333.3
MOVJ C00552 BC00552 VJ=20.00
MOVJ C00553 BC00553 VJ=30.00
MOVJ C00554 BC00554 VJ=30.00
MOVJ C00555 BC00555 VJ=30.00
MOVJ C00556 BC00556 VJ=30.00
'**********************
'W54B
'**********************
SFTON P0359
MOVL C00557 BC00557 V=250.0
MOVL C00558 BC00558 V=83.3 PL=0
SFTOF
MACRO1 MJ#(0) ARGF10
ARCON
SFTON P0360
MOVL C00559 BC00559 V=10.8
ARCOF
MOVL C00560 BC00560 V=333.3
SFTOF
MOVJ C00561 BC00561 VJ=30.00
MOVJ C00562 BC00562 VJ=30.00
MOVJ C00563 BC00563 VJ=30.00
MOVJ C00564 BC00564 VJ=40.00
MOVJ C00565 BC00565 VJ=40.00
MOVJ C00566 BC00566 VJ=10.00
MOVJ C00567 BC00567 VJ=10.00
MOVJ C00568 BC00568 VJ=10.00
MOVJ C00569 BC00569 VJ=15.00
MOVJ C00570 BC00570 VJ=15.00
MOVJ C00571 BC00571 VJ=15.00
MOVJ C00572 BC00572 VJ=15.00
'**********************
'W55A
'**********************
SFTON P0311
MOVL C00573 BC00573 V=166.7 PL=0
SFTOF
MACRO1 MJ#(0) ARGF10
ARCON
SFTON P0312
MOVL C00574 BC00574 V=10.8
MOVL C00575 BC00575 V=10.8
ARCOF
SFTOF
MOVL C00576 BC00576 V=150.0
MOVJ C00577 BC00577 VJ=10.00
MOVJ C00578 BC00578 VJ=10.00
MOVJ C00579 BC00579 VJ=10.00
MOVJ C00580 BC00580 VJ=10.00
MOVJ C00581 BC00581 VJ=10.00
MOVJ C00582 BC00582 VJ=10.00
MOVJ C00583 BC00583 VJ=30.00
MOVJ C00584 BC00584 VJ=30.00
MOVJ C00585 BC00585 VJ=20.00
MOVJ C00586 BC00586 VJ=30.00
MOVJ C00587 BC00587 VJ=20.00
MOVJ C00588 BC00588 VJ=20.00
MOVJ C00589 BC00589 VJ=30.00
MOVJ C00590 BC00590 VJ=20.00
MOVJ C00591 BC00591 VJ=20.00
'**********************
'W55B
'**********************
SFTON P0350
MOVL C00592 BC00592 V=333.3
MOVL C00593 BC00593 V=166.7 PL=0
SFTOF
MACRO1 MJ#(0) ARGF10
ARCON
SFTON P0349
MOVL C00594 BC00594 V=10.8
MOVL C00595 BC00595 V=10.8
ARCOF
SFTOF
MOVL C00596 BC00596 V=66.7
MOVJ C00597 BC00597 VJ=10.00
MOVJ C00598 BC00598 VJ=20.00
MOVJ C00599 BC00599 VJ=20.00
MOVJ C00600 BC00600 VJ=20.00
MOVJ C00601 BC00601 VJ=30.00
MOVJ C00602 BC00602 VJ=50.00
MOVJ C00603 BC00603 VJ=50.00
MOVJ C00604 BC00604 VJ=40.00
MOVJ C00605 BC00605 VJ=20.00
'**********************
'W56A
'**********************
SFTON P0308
MOVL C00606 BC00606 V=333.3
MOVL C00607 BC00607 V=166.7 PL=0
SFTOF
MACRO1 MJ#(0) ARGF10
ARCON
SFTON P0307
MOVL C00608 BC00608 V=10.8
ARCOF
SFTOF
MOVL C00609 BC00609 V=333.3
MOVJ C00610 BC00610 VJ=20.00
MOVJ C00611 BC00611 VJ=30.00
MOVJ C00612 BC00612 VJ=30.00
MOVJ C00613 BC00613 VJ=30.00
'**********************
'W56B
'**********************
SFTON P0353
MOVL C00614 BC00614 V=250.0
MOVL C00615 BC00615 V=166.7 PL=0
SFTOF
MACRO1 MJ#(0) ARGF10
ARCON
SFTON P0354
MOVL C00616 BC00616 V=10.8
ARCOF
SFTOF
MOVL C00617 BC00617 V=333.3
MOVJ C00618 BC00618 VJ=30.00
MOVJ C00619 BC00619 VJ=30.00
MOVJ C00620 BC00620 VJ=30.00
CALL JOB:MOVE_OUT_OF_TUNNEL
END
